// TwinCAT 3 PLC project lfe_optics
// Title: lcls-plc-lfe-optics
// Company: SLAC
// ProjectVersion: 4.0.0
// ProgramVersion: 3.1.4022.7
// CompilerDefines: L
// libraries:
//   LCLS General, * (SLAC)
//   lcls2-cc-lib, * (SLAC)
//   Tc2_ControllerToolbox, * (Beckhoff Automation GmbH)
//   Tc2_MC2, * (Beckhoff Automation GmbH)
//   Tc2_SerialCom, * (Beckhoff Automation GmbH)
//   Tc2_Standard, * (Beckhoff Automation GmbH)
//   Tc2_System, * (Beckhoff Automation GmbH)
//   Tc2_Utilities, * (Beckhoff Automation GmbH)
//   Tc3_Module, * (Beckhoff Automation GmbH)
//   VisuDialogs, * (System)
//   lcls-twincat-motion,4.0.9,SLAC
//   lcls-twincat-optics,0.7.0,SLAC
//   PMPS,3.3.0,SLAC - LCLS
// project tree:
//   DUTs/ E_MR1L0_CoatingStates.TcDUT, E_MR2L0_CoatingStates.TcDUT
//   Version/ Global_Version.TcGVL
//   / GlobalTextList.TcGTLO (not stored), PiezoDriver.TcTTO, PlcTask.TcTTO, SerialIO.TcTTO (not stored), Visualization Manager.TcVMO (not stored)
//   GVLs/ GVL_COM_Buffers.TcGVL, GVL_M1L0.TcGVL, GVL_M1L0_Constants.TcGVL, GVL_M2L0.TcGVL, GVL_M2L0_Constants.TcGVL, GVL_PMPS.TcGVL, GVL_SerialIO.TcGVL, GVL_States.TcGVL
//   POUs/ Main.TcPOU, PRG_1_PlcTask.TcPOU, PRG_MR1L0_HOMS.TcPOU, PRG_MR2L0_HOMS.TcPOU, PRG_PMPS.TcPOU, PRG_SP1L0_DCCM.TcPOU, P_CoatingProtections.TcPOU
//   POUs/Serial Comm/ PiezoSerial.TcPOU, P_Serial_Com.TcPOU
// real-time tasks:
//   TASK PlcTask: cycle T#10ms, priority 20, ADS port 350
//   TASK PiezoDriver: cycle T#1ms, priority 3, ADS port 351
//   TASK SerialIO: cycle T#2ms, priority 1, ADS port 352
// motion (NC):
//   TASK NC-Task 1 SAF: cycle T#2ms, priority 4, ADS port 501
//   TASK NC-Task 1 SVB: cycle T#10ms, priority 8, ADS port 511
//   AXIS M1L0-Yup (id 1)
//     General: UnitName=um
//     Dynamic: Acceleration=200, Deceleration=200, DelayTime=0.008
//     Velo: Maximum=200
//     OtherSettings: AllowMotionCmdToSlave=true
//     encoder EncType=29
//       EncPara: ScaleFactorNumerator=0.001, Offset=-16171.8, MaxCount=#xffffffff, ReferenceSystem=1
//         SoftEndMinControl: Enable=true, Range=-12605.3
//         SoftEndMaxControl: Enable=true, Range=10852.77
//         Inc: RefSoftSyncMask=#x0000ffff
//     drive DrvType=24
//       DrvPara: Inverse=true
//         Analog: VeloReferenz=488.28125, ScaleFactorActTorque=0.1
//         TimeComp: TaskDelayCycles=1
//     controller CtrType=2
//       CtrPara: PriorControlFactor=1
//         PosDiffControl: Range=100
//         PID: PosKp=50, PosExtKp=10, DeadBandPosition=0.3
//         Observer: BandWidth=20
//   AXIS M1L0-Ydwn (id 2)
//     General: UnitName=um
//     Dynamic: Acceleration=200, Deceleration=200, DelayTime=0.008
//     Velo: Maximum=200
//     OtherSettings: AllowMotionCmdToSlave=true
//     encoder EncType=29
//       EncPara: ScaleFactorNumerator=0.001, Offset=-14866.9, MaxCount=#xffffffff, ReferenceSystem=1
//         SoftEndMinControl: Enable=true, Range=-12700.5
//         SoftEndMaxControl: Enable=true, Range=10957.45
//         Inc: RefSoftSyncMask=#x0000ffff
//     drive DrvType=24
//       DrvPara: Inverse=true
//         Analog: VeloReferenz=488.28125, ScaleFactorActTorque=0.1
//         TimeComp: TaskDelayCycles=1
//     controller CtrType=2
//       CtrPara: PriorControlFactor=1
//         PosDiffControl: Range=100
//         PID: PosKp=50, PosExtKp=10, DeadBandPosition=0.3
//         Observer: BandWidth=20
//   AXIS M1L0-Xup (id 3)
//     General: UnitName=um
//     Dynamic: Acceleration=2000, Deceleration=2000, DelayTime=0.008
//     Velo: Maximum=1000
//     OtherSettings: AllowMotionCmdToSlave=true
//     encoder EncType=29
//       EncPara: ScaleFactorNumerator=0.001, Offset=-24797.788, MaxCount=#xffffffff, ReferenceSystem=1
//         SoftEndMinControl: Enable=true, Range=-600
//         SoftEndMaxControl: Enable=true, Range=690
//         Inc: RefSoftSyncMask=#x0000ffff
//     drive DrvType=24
//       Analog: VeloReferenz=1220.703125, ScaleFactorActTorque=0.1
//       TimeComp: TaskDelayCycles=1
//     controller CtrType=2
//       CtrPara: PriorControlFactor=1
//         PosDiffControl: Range=100
//         PID: PosKp=50, PosExtKp=50, DeadBandPosition=0.4
//         Observer: BandWidth=20
//   AXIS M1L0-Xdwn (id 4)
//     General: UnitName=um
//     Dynamic: Acceleration=2000, Deceleration=2000, DelayTime=0.008
//     Velo: Maximum=1000
//     OtherSettings: AllowMotionCmdToSlave=true
//     encoder EncType=29
//       EncPara: ScaleFactorNumerator=0.001, Offset=-22825.528, MaxCount=#xffffffff, ReferenceSystem=1
//         SoftEndMinControl: Enable=true, Range=-600
//         SoftEndMaxControl: Enable=true, Range=690
//         Inc: RefSoftSyncMask=#x0000ffff
//     drive DrvType=24
//       DrvPara: Inverse=true
//         Analog: VeloReferenz=1220.703125, ScaleFactorActTorque=0.1
//         TimeComp: TaskDelayCycles=1
//     controller CtrType=2
//       CtrPara: PriorControlFactor=1
//         PosDiffControl: Range=100
//         PID: PosKp=50, PosExtKp=50, DeadBandPosition=0.4
//         Observer: BandWidth=20
//   AXIS M1L0-Pitch (id 5)
//     General: UnitName=urad
//     Dynamic: Acceleration=390, Deceleration=390, DelayTime=0.008
//     Velo: Maximum=150
//     OtherSettings: AllowMotionCmdToSlave=true
//     encoder EncType=29
//       EncPara: ScaleFactorNumerator=0.001949317739, Offset=-16765.03, MaxCount=#xffffffff, ReferenceSystem=1
//         FilterTime: TPos=0.2
//         SoftEndMinControl: Enable=true, Range=-182
//         SoftEndMaxControl: Enable=true, Range=120
//         Inc: RefSoftSyncMask=#x0000ffff
//     drive DrvType=24
//       Analog: VeloReferenz=371.8, ScaleFactorActTorque=0.1
//       TimeComp: TaskDelayCycles=1
//     controller CtrType=2
//       CtrPara: PriorControlFactor=1
//         PosDiffControl: Range=20
//         PID: PosKp=2, PosExtKp=1, DeadBandPosition=0.01
//         Observer: BandWidth=20
//   AXIS M1L0-Bender (id 6)
//     General: UnitName=um
//     Dynamic: Acceleration=150, Deceleration=150, DelayTime=0.008
//     Velo: Maximum=150
//     OtherSettings: AllowMotionCmdToSlave=true
//     encoder EncType=29
//       EncPara: ScaleFactorNumerator=0.001, Offset=-4270000.1, MaxCount=#xffffffff, ReferenceSystem=1
//         SoftEndMinControl: Enable=true, Range=-1100.1
//         SoftEndMaxControl: Enable=true, Range=8149.9
//         Inc: RefSoftSyncMask=#x0000ffff
//     drive DrvType=24
//       DrvPara: Inverse=true
//         Analog: VeloReferenz=195.3125, ScaleFactorActTorque=0.1
//         TimeComp: TaskDelayCycles=1
//     controller CtrType=2
//       CtrPara: PriorControlFactor=1
//         PID: PosKp=10, PosExtKp=0.001, PosExtVelo=0.9, DeadBandPosition=0.1
//         Observer: BandWidth=20
//   AXIS M2L0-Yup (id 7)
//     General: UnitName=um
//     Dynamic: Acceleration=200, Deceleration=200, DelayTime=0.008
//     Velo: Maximum=200
//     OtherSettings: AllowMotionCmdToSlave=true
//     encoder EncType=29
//       EncPara: ScaleFactorNumerator=0.001, Offset=-12018.2, MaxCount=#xffffffff, MaxCountHighDWord=#x0000001f
//         SoftEndMinControl: Enable=true, Range=-9518.2
//         SoftEndMaxControl: Enable=true, Range=7519.8
//         Inc: RefSoftSyncMask=#x0000ffff
//     drive DrvType=24
//       DrvPara: Inverse=true
//         Analog: VeloReferenz=488.28125, ScaleFactorActTorque=0.1
//         TimeComp: TaskDelayCycles=1
//     controller CtrType=2
//       CtrPara: PriorControlFactor=1
//         PosDiffControl: Range=100
//         PID: PosKp=20, PosExtKp=5, DeadBandPosition=0.4
//         Observer: BandWidth=20
//   AXIS M2L0-Ydwn (id 8)
//     General: UnitName=um
//     Dynamic: Acceleration=200, Deceleration=200, DelayTime=0.008
//     Velo: Maximum=200
//     OtherSettings: AllowMotionCmdToSlave=true
//     encoder EncType=29
//       EncPara: ScaleFactorNumerator=0.001, Offset=-15143.7, MaxCount=#xffffffff, MaxCountHighDWord=#x0000001f
//         SoftEndMinControl: Enable=true, Range=-9987.7
//         SoftEndMaxControl: Enable=true, Range=7561.3
//         Inc: RefSoftSyncMask=#x0000ffff
//     drive DrvType=24
//       DrvPara: Inverse=true
//         Analog: VeloReferenz=488.28125, ScaleFactorActTorque=0.1
//         TimeComp: TaskDelayCycles=1
//     controller CtrType=2
//       CtrPara: PriorControlFactor=1
//         PosDiffControl: Range=100
//         PID: PosKp=20, PosExtKp=5, DeadBandPosition=0.4
//         Observer: BandWidth=20
//   AXIS M2L0-Xup (id 9)
//     General: UnitName=um
//     Dynamic: Acceleration=2000, Deceleration=2000, DelayTime=0.008
//     Velo: Maximum=1000
//     OtherSettings: AllowMotionCmdToSlave=true
//     encoder EncType=29
//       EncPara: ScaleFactorNumerator=0.001, Offset=-25363.4, MaxCount=#xffffffff, MaxCountHighDWord=#x0000001f
//         SoftEndMinControl: Enable=true, Range=-1063.4
//         SoftEndMaxControl: Enable=true, Range=1000
//         Inc: RefSoftSyncMask=#x0000ffff
//     drive DrvType=24
//       Analog: VeloReferenz=1220.703125, ScaleFactorActTorque=0.1
//       TimeComp: TaskDelayCycles=1
//     controller CtrType=2
//       CtrPara: PriorControlFactor=1
//         PosDiffControl: Range=100
//         PID: PosKp=10, PosExtKp=1, DeadBandPosition=0.4
//         Observer: BandWidth=20
//   AXIS M2L0-Xdwn (id 10)
//     General: UnitName=um
//     Dynamic: Acceleration=2000, Deceleration=2000, DelayTime=0.008
//     Velo: Maximum=1000
//     OtherSettings: AllowMotionCmdToSlave=true
//     encoder EncType=29
//       EncPara: ScaleFactorNumerator=0.001, Offset=-24398.1, MaxCount=#xffffffff, MaxCountHighDWord=#x0000001f
//         SoftEndMinControl: Enable=true, Range=-1289.2
//         SoftEndMaxControl: Enable=true, Range=1100.1
//         Inc: RefSoftSyncMask=#x0000ffff
//     drive DrvType=24
//       DrvPara: Inverse=true
//         Analog: VeloReferenz=1220.703125, ScaleFactorActTorque=0.1
//         TimeComp: TaskDelayCycles=1
//     controller CtrType=2
//       CtrPara: PriorControlFactor=1
//         PosDiffControl: Range=100
//         PID: PosKp=10, PosExtKp=1, DeadBandPosition=0.4
//         Observer: BandWidth=20
//   AXIS M2L0-Pitch (id 11)
//     General: UnitName=urad
//     Dynamic: Acceleration=390, Deceleration=390
//     Velo: Maximum=150
//     OtherSettings: AllowMotionCmdToSlave=true
//     encoder EncType=29
//       EncPara: ScaleFactorNumerator=0.001949317739, Offset=-18462.6, MaxCount=#xffffffff, MaxCountHighDWord=#x0000001f
//         FilterTime: TPos=0.2
//         SoftEndMinControl: Enable=true, Range=-45.1
//         SoftEndMaxControl: Enable=true, Range=154.9
//         Inc: RefSoftSyncMask=#x0000ffff
//     drive DrvType=24
//       Analog: VeloReferenz=371.8, ScaleFactorActTorque=0.1
//       TimeComp: TaskDelayCycles=1
//     controller CtrType=2
//       CtrPara: PriorControlFactor=1
//         PosDiffControl: Range=20
//         PID: PosKp=2, PosExtKp=1, DeadBandPosition=0.01
//         Observer: BandWidth=20
//   AXIS M2L0-Bender (id 12)
//     General: UnitName=um
//     Dynamic: Acceleration=150, Deceleration=150, DelayTime=0.008
//     Velo: Maximum=150
//     OtherSettings: AllowMotionCmdToSlave=true
//     encoder EncType=29
//       EncPara: ScaleFactorNumerator=0.001, Offset=-4268979, MaxCount=#xffffffff
//         SoftEndMinControl: Enable=true, Range=-2
//         SoftEndMaxControl: Enable=true, Range=10762
//         Inc: RefSoftSyncMask=#x0000ffff
//     drive DrvType=24
//       DrvPara: Inverse=true
//         Analog: VeloReferenz=195.3125, ScaleFactorActTorque=0.1
//         TimeComp: TaskDelayCycles=1
//     controller CtrType=2
//       CtrPara: PriorControlFactor=1
//         PID: PosKp=10, PosExtKp=0.001, PosExtVelo=0.9, DeadBandPosition=0.1
//         Observer: BandWidth=20
//   AXIS SP1L0-TH1 (id 13)
//     General: UnitName=Degree
//     Dynamic: AccelerationMaximum=10, DecelerationMaximum=10, Acceleration=8.99313, Deceleration=8.99313, Jerk=27.7544, DelayTime=0.008
//     Velo: SlowManual=1, FastManual=2, Maximum=0.12
//     TargetPosControl: Range=0.001
//     OtherSettings: AllowMotionCmdToSlave=true, PulseDistancePos=0.5, PulseDistanceNeg=0.5
//     encoder EncType=29
//       EncPara: ScaleFactorNumerator=5.72957795, ScaleFactorDenominator=10000000, Offset=-11, MaxCount=#xffffffff, MaxCountHighDWord=#x0000001f
//         SoftEndMinControl: Enable=true, Range=-1
//         SoftEndMaxControl: Enable=true, Range=71
//         Inc: RefSoftSyncMask=#x0000ffff
//     drive DrvType=24
//       Analog: VeloReferenz=0.1275, TorqueSetpointScale=10, ScaleFactorActTorque=0.1
//       TimeComp: TaskDelayCycles=1
//     controller CtrType=3
//       CtrPara: PriorControlFactor=1
//         PosDiffControl: Range=0.05
//         PID: PosKp=10, PosTv=0.2, DeadBandPosition=0.0001
//         Observer: BandWidth=20
//   AXIS SP1L0-TH2 (id 14)
//     General: UnitName=Degree
//     Dynamic: AccelerationMaximum=10, DecelerationMaximum=10, Acceleration=9, Deceleration=9, Jerk=27.7, DelayTime=0.008
//     Velo: SlowManual=0.1, FastManual=0.3, Maximum=0.12
//     PositionAreaControl: Range=0.05
//     TargetPosControl: Range=0.0001
//     OtherSettings: AllowMotionCmdToSlave=true
//     encoder EncType=29
//       EncPara: ScaleFactorNumerator=5.72957795, ScaleFactorDenominator=10000000, Offset=-10.66, MaxCount=#xffffffff, MaxCountHighDWord=#x0000001f
//         SoftEndMinControl: Enable=true, Range=-1
//         SoftEndMaxControl: Enable=true, Range=71
//         Inc: RefSoftSyncMask=#x0000ffff
//     drive DrvType=24
//       DrvPara: Inverse=true
//         Analog: VeloReferenz=0.127500425, TorqueSetpointScale=10, ScaleFactorActTorque=0.1
//         TimeComp: TaskDelayCycles=1
//     controller CtrType=3
//       CtrPara: PriorControlFactor=1
//         PosDiffControl: Range=0.05
//         PID: PosKp=10, PosTv=0.2, DeadBandPosition=0.0001
//         Observer: BandWidth=20
//   AXIS SP1L0-Tx (id 15)
//     Dynamic: AccelerationMaximum=20, DecelerationMaximum=20, Acceleration=10, Deceleration=10, Jerk=100, DelayTime=0.008
//     Velo: SlowManual=0.3, FastManual=1, Maximum=1
//     PositionAreaControl: Range=0.2
//     TargetPosControl: Range=0.0005
//     OtherSettings: AllowMotionCmdToSlave=true, PulseDistancePos=1, PulseDistanceNeg=1
//     encoder EncType=29
//       EncPara: ScaleFactorNumerator=50, ScaleFactorDenominator=1000000, Offset=-29.5, MaxCount=#xffffffff, MaxCountHighDWord=#x0000001f
//         SoftEndMinControl: Enable=true, Range=-13
//         SoftEndMaxControl: Enable=true, Range=3
//         Inc: RefSoftSyncMask=#x0000ffff
//     drive DrvType=24
//       Analog: VeloReferenz=1, TorqueSetpointScale=10, ScaleFactorActTorque=0.1
//       TimeComp: TaskDelayCycles=1
//     controller CtrType=3
//       CtrPara: PriorControlFactor=1
//         PosDiffControl: Range=0.1
//         PID: PosKp=10, PosTv=0.2, DeadBandPosition=0.0001
//         Observer: BandWidth=20
//   AXIS SP1L0-Txd (id 16)
//     Dynamic: AccelerationMaximum=20, DecelerationMaximum=20, Acceleration=10, Deceleration=10, Jerk=100, DelayTime=0.008
//     Velo: SlowManual=0.075, FastManual=0.2, Maximum=2
//     PositionAreaControl: Range=0.01
//     TargetPosControl: Range=0.0001
//     OtherSettings: AllowMotionCmdToSlave=true, PulseDistancePos=0.05, PulseDistanceNeg=0.05
//     encoder EncType=29
//       EncPara: ScaleFactorNumerator=50, ScaleFactorDenominator=1000000, Offset=-6871908.2, MaxCount=#xffffffff, MaxCountHighDWord=#x0000001f
//         SoftEndMinControl: Enable=true, Range=-12
//         SoftEndMaxControl: Enable=true, Range=12
//         Inc: RefSoftSyncMask=#x0000ffff
//     drive DrvType=24
//       DrvPara: Inverse=true
//         Analog: VeloReferenz=10.668, TorqueSetpointScale=10, ScaleFactorActTorque=0.1
//         TimeComp: TaskDelayCycles=1
//     controller CtrType=3
//       CtrPara: PriorControlFactor=1
//         PosDiffControl: Range=0.15
//         PID: PosKp=4, PosTv=0.2, PosTd=1, DeadBandPosition=0.0001
//         Observer: BandWidth=20
//   AXIS SP1L0-Tyd (id 17)
//     Dynamic: AccelerationMaximum=20, DecelerationMaximum=20, Acceleration=10, Deceleration=10, Jerk=100, DelayTime=0.008
//     Velo: SlowManual=0.5, FastManual=1, Maximum=2
//     PositionAreaControl: Range=0.05
//     TargetPosControl: Range=0.05
//     OtherSettings: AllowMotionCmdToSlave=true
//     encoder EncType=29
//       EncPara: ScaleFactorNumerator=50, ScaleFactorDenominator=1000000, Offset=-6871872.92, MaxCount=#xffffffff, MaxCountHighDWord=#x0000001f
//         SoftEndMaxControl: Range=48
//         Inc: RefSoftSyncMask=#x0000ffff
//     drive DrvType=24
//       Analog: VeloReferenz=12.6999, TorqueSetpointScale=10, ScaleFactorActTorque=0.1
//       TimeComp: TaskDelayCycles=1
//     controller CtrType=3
//       CtrPara: PriorControlFactor=1
//         PosDiffControl: Range=0.25
//         PID: PosKp=15, PosTv=0.2, DeadBandPosition=0.01
//         Observer: BandWidth=20
// I/O:
//   DEVICE Device 1 (EtherCAT), AmsNetId 172.21.88.30.2.1
//     Term 1 (EK1200) [EK1200-5000 EtherCAT Power supply (2A E-Bus)]
//       PMPS_FFO
//       Term 3 (EL6070) [EL6070 1Ch. Licensing-Terminal]
//       PMPS_PRE [EL6695 EtherCAT Bridge terminal (Primary)]
//       Term 5 (EK1122) [EK1122 2 port EtherCAT junction]
//         Box 6 (CU1124) [CU1124 EtherCAT junction (4-ports)]
//           EK1100_SP1L0 [EK1100 EtherCAT Coupler (2A E-Bus)]
//             EL7047_SP1L0_th1 [EL7047 1Ch. Stepper motor output stage (50V, 5A)]
//             EL7047_SP1L0_th2 [EL7047 1Ch. Stepper motor output stage (50V, 5A)]
//             EL7047_SP1L0_tx [EL7047 1Ch. Stepper motor output stage (50V, 5A)]
//             EL7047_SP1L0_txd [EL7047 1Ch. Stepper motor output stage (50V, 5A)]
//             EL7047_SP1L0_tyd [EL7047 1Ch. Stepper motor output stage (50V, 5A)]
//             EL5042_SP1L0_th1_th2 [EL5042 2Ch. BiSS-C Encoder]
//             EL5042_SP1L0_tx_txd [EL5042 2Ch. BiSS-C Encoder]
//             EL5042_SP1L0_tyd [EL5042 2Ch. BiSS-C Encoder]
//             EL1008_SP1L0_STO_DI [EL1008 8Ch. Dig. Input 24V, 3ms]
//             EL2008_SP1L0_DO [EL2008 8Ch. Dig. Output 24V, 0.5A]
//             EL3054_SP1L0_AI [EL3054 4Ch. Ana. Input 4-20mA]
//             EL9011_SP1L0 [EL9011 End Terminal]
//           EK1100_M2L0 [EK1100 EtherCAT Coupler (2A E-Bus)]
//             EL7041-1000_M2L0_Xup [EL7041-1000 1Ch. Stepper motor output stage (50V, 5A, standard)]
//             EL7041-1000_M2L0_Xdwn [EL7041-1000 1Ch. Stepper motor output stage (50V, 5A, standard)]
//             EL7041-1000_M2L0_Yup [EL7041-1000 1Ch. Stepper motor output stage (50V, 5A, standard)]
//             EL7041-1000_M2L0_Ydwn [EL7041-1000 1Ch. Stepper motor output stage (50V, 5A, standard)]
//             EL7041-1000_M2L0_PitchCoarse [EL7041-1000 1Ch. Stepper motor output stage (50V, 5A, standard)]
//             EL7041-1000_M2L0_Bender [EL7041-1000 1Ch. Stepper motor output stage (50V, 5A, standard)]
//             EL6001_M2L0_PitchFine [EL6001 Interface (RS232)]
//             EL5042_M2L0_Xupdwn [EL5042 2Ch. BiSS-C Encoder]
//             EL5042_M2L0_Yupdwn [EL5042 2Ch. BiSS-C Encoder]
//             EL5042_M2L0_PitchBender [EL5042 2Ch. BiSS-C Encoder]
//             EL1004_M2L0_STO [EL1004 4Ch. Dig. Input 24V, 3ms]
//             EL3054_M2L0_FWM_PRSM [EL3054 4Ch. Ana. Input 4-20mA]
//             EL9505_M2L0_BenderLims [EL9505 Power supply terminal 5V]
//             Term 33 (EL9011) [EL9011 End Terminal]
//           EP2008-0001_M1M2_VCV
//         EK1100_M1L0 [EK1100 EtherCAT Coupler (2A E-Bus)]
//           EL7041-1000_M1L0_Xup [EL7041-1000 1Ch. Stepper motor output stage (50V, 5A, standard)]
//           EL7041-1000_M1L0_Xdwn
//           EL7041-1000_M1L0_Yup [EL7041-1000 1Ch. Stepper motor output stage (50V, 5A, standard)]
//           EL7041-1000_M1L0_Ydwn [EL7041-1000 1Ch. Stepper motor output stage (50V, 5A, standard)]
//           EL7041-1000_M1L0_PitchCoarse [EL7041-1000 1Ch. Stepper motor output stage (50V, 5A, standard)]
//           EL7041-1000_M1L0_Bender
//           EL6001_M1L0_PitchFine
//           EL5042_M1L0_Xupdwn
//           EL5042_M1L0_Yupdwn
//           EL5042_M1L0_PitchBender [EL5042 2Ch. BiSS-C Encoder]
//           EL1004_M1L0_STO
//           EL3054_M1L0_FWM_PRSM
//           EL9505_M1L0_BenderLims
//           Term 32 (EL9011)
// variable links:
//   (this object) <-> Device 1 (EtherCAT)/Term 1 (EK1200)/Term 5 (EK1122)/EK1100_M1L0/EL5042_M1L0_Yupdwn
//     Enc/Inputs/In/nComState @bit 1 <-> WcState/InputToggle
//     Enc/Inputs/In/nComState <-> WcState/WcState
//     Enc/Inputs/In/nDataIn1 <-> FB Inputs Channel 1/Position
//     Enc/Inputs/In/nDataIn1 <-> FB Inputs Channel 2/Position
//     Enc/Inputs/In/nState1 @bit 12 <-> FB Inputs Channel 1/Status/Diag
//     Enc/Inputs/In/nState1 @bit 12 <-> FB Inputs Channel 2/Status/Diag
//     Enc/Inputs/In/nState1 @bit 1 <-> FB Inputs Channel 1/Status/Error
//     Enc/Inputs/In/nState1 @bit 1 <-> FB Inputs Channel 2/Status/Error
//     Enc/Inputs/In/nState1 @bit 14 <-> FB Inputs Channel 1/Status/Input cycle counter
//     Enc/Inputs/In/nState1 @bit 14 <-> FB Inputs Channel 2/Status/Input cycle counter
//     Enc/Inputs/In/nState1 @bit 2 <-> FB Inputs Channel 1/Status/Ready
//     Enc/Inputs/In/nState1 @bit 2 <-> FB Inputs Channel 2/Status/Ready
//     Enc/Inputs/In/nState1 @bit 13 <-> FB Inputs Channel 1/Status/TxPDO State
//     Enc/Inputs/In/nState1 @bit 13 <-> FB Inputs Channel 2/Status/TxPDO State
//     Enc/Inputs/In/nState1 <-> FB Inputs Channel 1/Status/Warning
//     Enc/Inputs/In/nState1 <-> FB Inputs Channel 2/Status/Warning
//   (this object) <-> Device 1 (EtherCAT)/Term 1 (EK1200)/Term 5 (EK1122)/EK1100_M1L0/EL7041-1000_M1L0_Yup
//     Drive/Inputs/In/nState1 @bit 3 <-> STM Status/Status/Error
//     Drive/Inputs/In/nState1 @bit 5 <-> STM Status/Status/Moving negative
//     Drive/Inputs/In/nState1 @bit 4 <-> STM Status/Status/Moving positive
//     Drive/Inputs/In/nState1 @bit 1 <-> STM Status/Status/Ready
//     Drive/Inputs/In/nState1 <-> STM Status/Status/Ready to enable
//     Drive/Inputs/In/nState1 @bit 6 <-> STM Status/Status/Torque reduced
//     Drive/Inputs/In/nState1 @bit 2 <-> STM Status/Status/Warning
//     Drive/Inputs/In/nState2 @bit 3 <-> STM Status/Status/Digital input 1
//     Drive/Inputs/In/nState2 @bit 4 <-> STM Status/Status/Digital input 2
//     Drive/Inputs/In/nState2 @bit 5 <-> STM Status/Status/Sync error
//     Drive/Inputs/In/nState2 @bit 7 <-> STM Status/Status/TxPDO Toggle
//     Drive/Inputs/In/nState4 @bit 1 <-> WcState/InputToggle
//     Drive/Inputs/In/nState4 <-> WcState/WcState
//     Drive/Outputs/Out/nCtrl1 <-> STM Control/Control/Enable
//     Drive/Outputs/Out/nCtrl1 @bit 2 <-> STM Control/Control/Reduce torque
//     Drive/Outputs/Out/nCtrl1 @bit 1 <-> STM Control/Control/Reset
//     Drive/Outputs/Out/nDataOut2[0] <-> STM Velocity/Velocity
//   (this object) <-> Device 1 (EtherCAT)/Term 1 (EK1200)/Term 5 (EK1122)/EK1100_M1L0/EL7041-1000_M1L0_Ydwn
//     Drive/Inputs/In/nState1 @bit 3 <-> STM Status/Status/Error
//     Drive/Inputs/In/nState1 @bit 5 <-> STM Status/Status/Moving negative
//     Drive/Inputs/In/nState1 @bit 4 <-> STM Status/Status/Moving positive
//     Drive/Inputs/In/nState1 @bit 1 <-> STM Status/Status/Ready
//     Drive/Inputs/In/nState1 <-> STM Status/Status/Ready to enable
//     Drive/Inputs/In/nState1 @bit 6 <-> STM Status/Status/Torque reduced
//     Drive/Inputs/In/nState1 @bit 2 <-> STM Status/Status/Warning
//     Drive/Inputs/In/nState2 @bit 3 <-> STM Status/Status/Digital input 1
//     Drive/Inputs/In/nState2 @bit 4 <-> STM Status/Status/Digital input 2
//     Drive/Inputs/In/nState2 @bit 5 <-> STM Status/Status/Sync error
//     Drive/Inputs/In/nState2 @bit 7 <-> STM Status/Status/TxPDO Toggle
//     Drive/Inputs/In/nState4 @bit 1 <-> WcState/InputToggle
//     Drive/Inputs/In/nState4 <-> WcState/WcState
//     Drive/Outputs/Out/nCtrl1 <-> STM Control/Control/Enable
//     Drive/Outputs/Out/nCtrl1 @bit 2 <-> STM Control/Control/Reduce torque
//     Drive/Outputs/Out/nCtrl1 @bit 1 <-> STM Control/Control/Reset
//     Drive/Outputs/Out/nDataOut2[0] <-> STM Velocity/Velocity
//   (this object) <-> Device 1 (EtherCAT)/Term 1 (EK1200)/Term 5 (EK1122)/EK1100_M1L0/EL5042_M1L0_Xupdwn
//     Enc/Inputs/In/nComState @bit 1 <-> WcState/InputToggle
//     Enc/Inputs/In/nComState <-> WcState/WcState
//     Enc/Inputs/In/nDataIn1 <-> FB Inputs Channel 1/Position
//     Enc/Inputs/In/nDataIn1 <-> FB Inputs Channel 2/Position
//     Enc/Inputs/In/nState1 @bit 12 <-> FB Inputs Channel 1/Status/Diag
//     Enc/Inputs/In/nState1 @bit 12 <-> FB Inputs Channel 2/Status/Diag
//     Enc/Inputs/In/nState1 @bit 1 <-> FB Inputs Channel 1/Status/Error
//     Enc/Inputs/In/nState1 @bit 1 <-> FB Inputs Channel 2/Status/Error
//     Enc/Inputs/In/nState1 @bit 14 <-> FB Inputs Channel 1/Status/Input cycle counter
//     Enc/Inputs/In/nState1 @bit 14 <-> FB Inputs Channel 2/Status/Input cycle counter
//     Enc/Inputs/In/nState1 @bit 2 <-> FB Inputs Channel 1/Status/Ready
//     Enc/Inputs/In/nState1 @bit 2 <-> FB Inputs Channel 2/Status/Ready
//     Enc/Inputs/In/nState1 @bit 13 <-> FB Inputs Channel 1/Status/TxPDO State
//     Enc/Inputs/In/nState1 @bit 13 <-> FB Inputs Channel 2/Status/TxPDO State
//     Enc/Inputs/In/nState1 <-> FB Inputs Channel 1/Status/Warning
//     Enc/Inputs/In/nState1 <-> FB Inputs Channel 2/Status/Warning
//   (this object) <-> Device 1 (EtherCAT)/Term 1 (EK1200)/Term 5 (EK1122)/EK1100_M1L0/EL7041-1000_M1L0_Xup
//     Drive/Inputs/In/nState1 @bit 3 <-> STM Status/Status/Error
//     Drive/Inputs/In/nState1 @bit 5 <-> STM Status/Status/Moving negative
//     Drive/Inputs/In/nState1 @bit 4 <-> STM Status/Status/Moving positive
//     Drive/Inputs/In/nState1 @bit 1 <-> STM Status/Status/Ready
//     Drive/Inputs/In/nState1 <-> STM Status/Status/Ready to enable
//     Drive/Inputs/In/nState1 @bit 6 <-> STM Status/Status/Torque reduced
//     Drive/Inputs/In/nState1 @bit 2 <-> STM Status/Status/Warning
//     Drive/Inputs/In/nState2 @bit 3 <-> STM Status/Status/Digital input 1
//     Drive/Inputs/In/nState2 @bit 4 <-> STM Status/Status/Digital input 2
//     Drive/Inputs/In/nState2 @bit 5 <-> STM Status/Status/Sync error
//     Drive/Inputs/In/nState2 @bit 7 <-> STM Status/Status/TxPDO Toggle
//     Drive/Inputs/In/nState4 @bit 1 <-> WcState/InputToggle
//     Drive/Inputs/In/nState4 <-> WcState/WcState
//     Drive/Outputs/Out/nCtrl1 <-> STM Control/Control/Enable
//     Drive/Outputs/Out/nCtrl1 @bit 2 <-> STM Control/Control/Reduce torque
//     Drive/Outputs/Out/nCtrl1 @bit 1 <-> STM Control/Control/Reset
//     Drive/Outputs/Out/nDataOut2[0] <-> STM Velocity/Velocity
//   (this object) <-> Device 1 (EtherCAT)/Term 1 (EK1200)/Term 5 (EK1122)/EK1100_M1L0/EL7041-1000_M1L0_Xdwn
//     Drive/Inputs/In/nState1 @bit 3 <-> STM Status/Status/Error
//     Drive/Inputs/In/nState1 @bit 5 <-> STM Status/Status/Moving negative
//     Drive/Inputs/In/nState1 @bit 4 <-> STM Status/Status/Moving positive
//     Drive/Inputs/In/nState1 @bit 1 <-> STM Status/Status/Ready
//     Drive/Inputs/In/nState1 <-> STM Status/Status/Ready to enable
//     Drive/Inputs/In/nState1 @bit 6 <-> STM Status/Status/Torque reduced
//     Drive/Inputs/In/nState1 @bit 2 <-> STM Status/Status/Warning
//     Drive/Inputs/In/nState2 @bit 3 <-> STM Status/Status/Digital input 1
//     Drive/Inputs/In/nState2 @bit 4 <-> STM Status/Status/Digital input 2
//     Drive/Inputs/In/nState2 @bit 5 <-> STM Status/Status/Sync error
//     Drive/Inputs/In/nState2 @bit 7 <-> STM Status/Status/TxPDO Toggle
//     Drive/Inputs/In/nState4 @bit 1 <-> WcState/InputToggle
//     Drive/Inputs/In/nState4 <-> WcState/WcState
//     Drive/Outputs/Out/nCtrl1 <-> STM Control/Control/Enable
//     Drive/Outputs/Out/nCtrl1 @bit 2 <-> STM Control/Control/Reduce torque
//     Drive/Outputs/Out/nCtrl1 @bit 1 <-> STM Control/Control/Reset
//     Drive/Outputs/Out/nDataOut2[0] <-> STM Velocity/Velocity
//   (this object) <-> Device 1 (EtherCAT)/Term 1 (EK1200)/Term 5 (EK1122)/EK1100_M1L0/EL5042_M1L0_PitchBender
//     Enc/Inputs/In/nComState @bit 1 <-> WcState/InputToggle
//     Enc/Inputs/In/nComState <-> WcState/WcState
//     Enc/Inputs/In/nDataIn1 <-> FB Inputs Channel 1/Position
//     Enc/Inputs/In/nDataIn1 <-> FB Inputs Channel 2/Position
//     Enc/Inputs/In/nState1 @bit 12 <-> FB Inputs Channel 1/Status/Diag
//     Enc/Inputs/In/nState1 @bit 12 <-> FB Inputs Channel 2/Status/Diag
//     Enc/Inputs/In/nState1 @bit 1 <-> FB Inputs Channel 1/Status/Error
//     Enc/Inputs/In/nState1 @bit 1 <-> FB Inputs Channel 2/Status/Error
//     Enc/Inputs/In/nState1 @bit 14 <-> FB Inputs Channel 1/Status/Input cycle counter
//     Enc/Inputs/In/nState1 @bit 14 <-> FB Inputs Channel 2/Status/Input cycle counter
//     Enc/Inputs/In/nState1 @bit 2 <-> FB Inputs Channel 1/Status/Ready
//     Enc/Inputs/In/nState1 @bit 2 <-> FB Inputs Channel 2/Status/Ready
//     Enc/Inputs/In/nState1 @bit 13 <-> FB Inputs Channel 1/Status/TxPDO State
//     Enc/Inputs/In/nState1 @bit 13 <-> FB Inputs Channel 2/Status/TxPDO State
//     Enc/Inputs/In/nState1 <-> FB Inputs Channel 1/Status/Warning
//     Enc/Inputs/In/nState1 <-> FB Inputs Channel 2/Status/Warning
//   (this object) <-> Device 1 (EtherCAT)/Term 1 (EK1200)/Term 5 (EK1122)/EK1100_M1L0/EL7041-1000_M1L0_PitchCoarse
//     Drive/Inputs/In/nState1 @bit 3 <-> STM Status/Status/Error
//     Drive/Inputs/In/nState1 @bit 5 <-> STM Status/Status/Moving negative
//     Drive/Inputs/In/nState1 @bit 4 <-> STM Status/Status/Moving positive
//     Drive/Inputs/In/nState1 @bit 1 <-> STM Status/Status/Ready
//     Drive/Inputs/In/nState1 <-> STM Status/Status/Ready to enable
//     Drive/Inputs/In/nState1 @bit 6 <-> STM Status/Status/Torque reduced
//     Drive/Inputs/In/nState1 @bit 2 <-> STM Status/Status/Warning
//     Drive/Inputs/In/nState2 @bit 3 <-> STM Status/Status/Digital input 1
//     Drive/Inputs/In/nState2 @bit 4 <-> STM Status/Status/Digital input 2
//     Drive/Inputs/In/nState2 @bit 5 <-> STM Status/Status/Sync error
//     Drive/Inputs/In/nState2 @bit 7 <-> STM Status/Status/TxPDO Toggle
//     Drive/Inputs/In/nState4 @bit 1 <-> WcState/InputToggle
//     Drive/Inputs/In/nState4 <-> WcState/WcState
//     Drive/Outputs/Out/nCtrl1 <-> STM Control/Control/Enable
//     Drive/Outputs/Out/nCtrl1 @bit 2 <-> STM Control/Control/Reduce torque
//     Drive/Outputs/Out/nCtrl1 @bit 1 <-> STM Control/Control/Reset
//     Drive/Outputs/Out/nDataOut2[0] <-> STM Velocity/Velocity
//   (this object) <-> Device 1 (EtherCAT)/Term 1 (EK1200)/Term 5 (EK1122)/EK1100_M1L0/EL7041-1000_M1L0_Bender
//     Drive/Inputs/In/nState1 @bit 3 <-> STM Status/Status/Error
//     Drive/Inputs/In/nState1 @bit 5 <-> STM Status/Status/Moving negative
//     Drive/Inputs/In/nState1 @bit 4 <-> STM Status/Status/Moving positive
//     Drive/Inputs/In/nState1 @bit 1 <-> STM Status/Status/Ready
//     Drive/Inputs/In/nState1 <-> STM Status/Status/Ready to enable
//     Drive/Inputs/In/nState1 @bit 6 <-> STM Status/Status/Torque reduced
//     Drive/Inputs/In/nState1 @bit 2 <-> STM Status/Status/Warning
//     Drive/Inputs/In/nState2 @bit 3 <-> STM Status/Status/Digital input 1
//     Drive/Inputs/In/nState2 @bit 4 <-> STM Status/Status/Digital input 2
//     Drive/Inputs/In/nState2 @bit 5 <-> STM Status/Status/Sync error
//     Drive/Inputs/In/nState2 @bit 7 <-> STM Status/Status/TxPDO Toggle
//     Drive/Inputs/In/nState4 @bit 1 <-> WcState/InputToggle
//     Drive/Inputs/In/nState4 <-> WcState/WcState
//     Drive/Outputs/Out/nCtrl1 <-> STM Control/Control/Enable
//     Drive/Outputs/Out/nCtrl1 @bit 2 <-> STM Control/Control/Reduce torque
//     Drive/Outputs/Out/nCtrl1 @bit 1 <-> STM Control/Control/Reset
//     Drive/Outputs/Out/nDataOut2[0] <-> STM Velocity/Velocity
//   (this object) <-> Device 1 (EtherCAT)/Term 1 (EK1200)/Term 5 (EK1122)/Box 6 (CU1124)/EK1100_M2L0/EL5042_M2L0_Yupdwn
//     Enc/Inputs/In/nComState @bit 1 <-> WcState/InputToggle
//     Enc/Inputs/In/nComState <-> WcState/WcState
//     Enc/Inputs/In/nDataIn1 <-> FB Inputs Channel 1/Position
//     Enc/Inputs/In/nDataIn1 <-> FB Inputs Channel 2/Position
//     Enc/Inputs/In/nState1 @bit 12 <-> FB Inputs Channel 1/Status/Diag
//     Enc/Inputs/In/nState1 @bit 12 <-> FB Inputs Channel 2/Status/Diag
//     Enc/Inputs/In/nState1 @bit 1 <-> FB Inputs Channel 1/Status/Error
//     Enc/Inputs/In/nState1 @bit 1 <-> FB Inputs Channel 2/Status/Error
//     Enc/Inputs/In/nState1 @bit 14 <-> FB Inputs Channel 1/Status/Input cycle counter
//     Enc/Inputs/In/nState1 @bit 14 <-> FB Inputs Channel 2/Status/Input cycle counter
//     Enc/Inputs/In/nState1 @bit 2 <-> FB Inputs Channel 1/Status/Ready
//     Enc/Inputs/In/nState1 @bit 2 <-> FB Inputs Channel 2/Status/Ready
//     Enc/Inputs/In/nState1 @bit 13 <-> FB Inputs Channel 1/Status/TxPDO State
//     Enc/Inputs/In/nState1 @bit 13 <-> FB Inputs Channel 2/Status/TxPDO State
//     Enc/Inputs/In/nState1 <-> FB Inputs Channel 1/Status/Warning
//     Enc/Inputs/In/nState1 <-> FB Inputs Channel 2/Status/Warning
//   (this object) <-> Device 1 (EtherCAT)/Term 1 (EK1200)/Term 5 (EK1122)/Box 6 (CU1124)/EK1100_M2L0/EL7041-1000_M2L0_Yup
//     Drive/Inputs/In/nState1 @bit 3 <-> STM Status/Status/Error
//     Drive/Inputs/In/nState1 @bit 5 <-> STM Status/Status/Moving negative
//     Drive/Inputs/In/nState1 @bit 4 <-> STM Status/Status/Moving positive
//     Drive/Inputs/In/nState1 @bit 1 <-> STM Status/Status/Ready
//     Drive/Inputs/In/nState1 <-> STM Status/Status/Ready to enable
//     Drive/Inputs/In/nState1 @bit 6 <-> STM Status/Status/Torque reduced
//     Drive/Inputs/In/nState1 @bit 2 <-> STM Status/Status/Warning
//     Drive/Inputs/In/nState2 @bit 3 <-> STM Status/Status/Digital input 1
//     Drive/Inputs/In/nState2 @bit 4 <-> STM Status/Status/Digital input 2
//     Drive/Inputs/In/nState2 @bit 5 <-> STM Status/Status/Sync error
//     Drive/Inputs/In/nState2 @bit 7 <-> STM Status/Status/TxPDO Toggle
//     Drive/Inputs/In/nState4 @bit 1 <-> WcState/InputToggle
//     Drive/Inputs/In/nState4 <-> WcState/WcState
//     Drive/Outputs/Out/nCtrl1 <-> STM Control/Control/Enable
//     Drive/Outputs/Out/nCtrl1 @bit 2 <-> STM Control/Control/Reduce torque
//     Drive/Outputs/Out/nCtrl1 @bit 1 <-> STM Control/Control/Reset
//     Drive/Outputs/Out/nDataOut2[0] <-> STM Velocity/Velocity
//   (this object) <-> Device 1 (EtherCAT)/Term 1 (EK1200)/Term 5 (EK1122)/Box 6 (CU1124)/EK1100_M2L0/EL7041-1000_M2L0_Ydwn
//     Drive/Inputs/In/nState1 @bit 3 <-> STM Status/Status/Error
//     Drive/Inputs/In/nState1 @bit 5 <-> STM Status/Status/Moving negative
//     Drive/Inputs/In/nState1 @bit 4 <-> STM Status/Status/Moving positive
//     Drive/Inputs/In/nState1 @bit 1 <-> STM Status/Status/Ready
//     Drive/Inputs/In/nState1 <-> STM Status/Status/Ready to enable
//     Drive/Inputs/In/nState1 @bit 6 <-> STM Status/Status/Torque reduced
//     Drive/Inputs/In/nState1 @bit 2 <-> STM Status/Status/Warning
//     Drive/Inputs/In/nState2 @bit 3 <-> STM Status/Status/Digital input 1
//     Drive/Inputs/In/nState2 @bit 4 <-> STM Status/Status/Digital input 2
//     Drive/Inputs/In/nState2 @bit 5 <-> STM Status/Status/Sync error
//     Drive/Inputs/In/nState2 @bit 7 <-> STM Status/Status/TxPDO Toggle
//     Drive/Inputs/In/nState4 @bit 1 <-> WcState/InputToggle
//     Drive/Inputs/In/nState4 <-> WcState/WcState
//     Drive/Outputs/Out/nCtrl1 <-> STM Control/Control/Enable
//     Drive/Outputs/Out/nCtrl1 @bit 2 <-> STM Control/Control/Reduce torque
//     Drive/Outputs/Out/nCtrl1 @bit 1 <-> STM Control/Control/Reset
//     Drive/Outputs/Out/nDataOut2[0] <-> STM Velocity/Velocity
//   (this object) <-> Device 1 (EtherCAT)/Term 1 (EK1200)/Term 5 (EK1122)/Box 6 (CU1124)/EK1100_M2L0/EL5042_M2L0_Xupdwn
//     Enc/Inputs/In/nComState @bit 1 <-> WcState/InputToggle
//     Enc/Inputs/In/nComState <-> WcState/WcState
//     Enc/Inputs/In/nDataIn1 <-> FB Inputs Channel 1/Position
//     Enc/Inputs/In/nDataIn1 <-> FB Inputs Channel 2/Position
//     Enc/Inputs/In/nState1 @bit 12 <-> FB Inputs Channel 1/Status/Diag
//     Enc/Inputs/In/nState1 @bit 12 <-> FB Inputs Channel 2/Status/Diag
//     Enc/Inputs/In/nState1 @bit 1 <-> FB Inputs Channel 1/Status/Error
//     Enc/Inputs/In/nState1 @bit 1 <-> FB Inputs Channel 2/Status/Error
//     Enc/Inputs/In/nState1 @bit 14 <-> FB Inputs Channel 1/Status/Input cycle counter
//     Enc/Inputs/In/nState1 @bit 14 <-> FB Inputs Channel 2/Status/Input cycle counter
//     Enc/Inputs/In/nState1 @bit 2 <-> FB Inputs Channel 1/Status/Ready
//     Enc/Inputs/In/nState1 @bit 2 <-> FB Inputs Channel 2/Status/Ready
//     Enc/Inputs/In/nState1 @bit 13 <-> FB Inputs Channel 1/Status/TxPDO State
//     Enc/Inputs/In/nState1 @bit 13 <-> FB Inputs Channel 2/Status/TxPDO State
//     Enc/Inputs/In/nState1 <-> FB Inputs Channel 1/Status/Warning
//     Enc/Inputs/In/nState1 <-> FB Inputs Channel 2/Status/Warning
//   (this object) <-> Device 1 (EtherCAT)/Term 1 (EK1200)/Term 5 (EK1122)/Box 6 (CU1124)/EK1100_M2L0/EL7041-1000_M2L0_Xup
//     Drive/Inputs/In/nState1 @bit 3 <-> STM Status/Status/Error
//     Drive/Inputs/In/nState1 @bit 5 <-> STM Status/Status/Moving negative
//     Drive/Inputs/In/nState1 @bit 4 <-> STM Status/Status/Moving positive
//     Drive/Inputs/In/nState1 @bit 1 <-> STM Status/Status/Ready
//     Drive/Inputs/In/nState1 <-> STM Status/Status/Ready to enable
//     Drive/Inputs/In/nState1 @bit 6 <-> STM Status/Status/Torque reduced
//     Drive/Inputs/In/nState1 @bit 2 <-> STM Status/Status/Warning
//     Drive/Inputs/In/nState2 @bit 3 <-> STM Status/Status/Digital input 1
//     Drive/Inputs/In/nState2 @bit 4 <-> STM Status/Status/Digital input 2
//     Drive/Inputs/In/nState2 @bit 5 <-> STM Status/Status/Sync error
//     Drive/Inputs/In/nState2 @bit 7 <-> STM Status/Status/TxPDO Toggle
//     Drive/Inputs/In/nState4 @bit 1 <-> WcState/InputToggle
//     Drive/Inputs/In/nState4 <-> WcState/WcState
//     Drive/Outputs/Out/nCtrl1 <-> STM Control/Control/Enable
//     Drive/Outputs/Out/nCtrl1 @bit 2 <-> STM Control/Control/Reduce torque
//     Drive/Outputs/Out/nCtrl1 @bit 1 <-> STM Control/Control/Reset
//     Drive/Outputs/Out/nDataOut2[0] <-> STM Velocity/Velocity
//   (this object) <-> Device 1 (EtherCAT)/Term 1 (EK1200)/Term 5 (EK1122)/Box 6 (CU1124)/EK1100_M2L0/EL7041-1000_M2L0_Xdwn
//     Drive/Inputs/In/nState1 @bit 3 <-> STM Status/Status/Error
//     Drive/Inputs/In/nState1 @bit 5 <-> STM Status/Status/Moving negative
//     Drive/Inputs/In/nState1 @bit 4 <-> STM Status/Status/Moving positive
//     Drive/Inputs/In/nState1 @bit 1 <-> STM Status/Status/Ready
//     Drive/Inputs/In/nState1 <-> STM Status/Status/Ready to enable
//     Drive/Inputs/In/nState1 @bit 6 <-> STM Status/Status/Torque reduced
//     Drive/Inputs/In/nState1 @bit 2 <-> STM Status/Status/Warning
//     Drive/Inputs/In/nState2 @bit 3 <-> STM Status/Status/Digital input 1
//     Drive/Inputs/In/nState2 @bit 4 <-> STM Status/Status/Digital input 2
//     Drive/Inputs/In/nState2 @bit 5 <-> STM Status/Status/Sync error
//     Drive/Inputs/In/nState2 @bit 7 <-> STM Status/Status/TxPDO Toggle
//     Drive/Inputs/In/nState4 @bit 1 <-> WcState/InputToggle
//     Drive/Inputs/In/nState4 <-> WcState/WcState
//     Drive/Outputs/Out/nCtrl1 <-> STM Control/Control/Enable
//     Drive/Outputs/Out/nCtrl1 @bit 2 <-> STM Control/Control/Reduce torque
//     Drive/Outputs/Out/nCtrl1 @bit 1 <-> STM Control/Control/Reset
//     Drive/Outputs/Out/nDataOut2[0] <-> STM Velocity/Velocity
//   (this object) <-> Device 1 (EtherCAT)/Term 1 (EK1200)/Term 5 (EK1122)/Box 6 (CU1124)/EK1100_M2L0/EL5042_M2L0_PitchBender
//     Enc/Inputs/In/nComState @bit 1 <-> WcState/InputToggle
//     Enc/Inputs/In/nComState <-> WcState/WcState
//     Enc/Inputs/In/nDataIn1 <-> FB Inputs Channel 1/Position
//     Enc/Inputs/In/nDataIn1 <-> FB Inputs Channel 2/Position
//     Enc/Inputs/In/nState1 @bit 12 <-> FB Inputs Channel 1/Status/Diag
//     Enc/Inputs/In/nState1 @bit 12 <-> FB Inputs Channel 2/Status/Diag
//     Enc/Inputs/In/nState1 @bit 1 <-> FB Inputs Channel 1/Status/Error
//     Enc/Inputs/In/nState1 @bit 1 <-> FB Inputs Channel 2/Status/Error
//     Enc/Inputs/In/nState1 @bit 14 <-> FB Inputs Channel 1/Status/Input cycle counter
//     Enc/Inputs/In/nState1 @bit 14 <-> FB Inputs Channel 2/Status/Input cycle counter
//     Enc/Inputs/In/nState1 @bit 2 <-> FB Inputs Channel 1/Status/Ready
//     Enc/Inputs/In/nState1 @bit 2 <-> FB Inputs Channel 2/Status/Ready
//     Enc/Inputs/In/nState1 @bit 13 <-> FB Inputs Channel 1/Status/TxPDO State
//     Enc/Inputs/In/nState1 @bit 13 <-> FB Inputs Channel 2/Status/TxPDO State
//     Enc/Inputs/In/nState1 <-> FB Inputs Channel 1/Status/Warning
//     Enc/Inputs/In/nState1 <-> FB Inputs Channel 2/Status/Warning
//   (this object) <-> Device 1 (EtherCAT)/Term 1 (EK1200)/Term 5 (EK1122)/Box 6 (CU1124)/EK1100_M2L0/EL7041-1000_M2L0_PitchCoarse
//     Drive/Inputs/In/nState1 @bit 3 <-> STM Status/Status/Error
//     Drive/Inputs/In/nState1 @bit 5 <-> STM Status/Status/Moving negative
//     Drive/Inputs/In/nState1 @bit 4 <-> STM Status/Status/Moving positive
//     Drive/Inputs/In/nState1 @bit 1 <-> STM Status/Status/Ready
//     Drive/Inputs/In/nState1 <-> STM Status/Status/Ready to enable
//     Drive/Inputs/In/nState1 @bit 6 <-> STM Status/Status/Torque reduced
//     Drive/Inputs/In/nState1 @bit 2 <-> STM Status/Status/Warning
//     Drive/Inputs/In/nState2 @bit 3 <-> STM Status/Status/Digital input 1
//     Drive/Inputs/In/nState2 @bit 4 <-> STM Status/Status/Digital input 2
//     Drive/Inputs/In/nState2 @bit 5 <-> STM Status/Status/Sync error
//     Drive/Inputs/In/nState2 @bit 7 <-> STM Status/Status/TxPDO Toggle
//     Drive/Inputs/In/nState4 @bit 1 <-> WcState/InputToggle
//     Drive/Inputs/In/nState4 <-> WcState/WcState
//     Drive/Outputs/Out/nCtrl1 <-> STM Control/Control/Enable
//     Drive/Outputs/Out/nCtrl1 @bit 2 <-> STM Control/Control/Reduce torque
//     Drive/Outputs/Out/nCtrl1 @bit 1 <-> STM Control/Control/Reset
//     Drive/Outputs/Out/nDataOut2[0] <-> STM Velocity/Velocity
//   (this object) <-> Device 1 (EtherCAT)/Term 1 (EK1200)/Term 5 (EK1122)/Box 6 (CU1124)/EK1100_M2L0/EL7041-1000_M2L0_Bender
//     Drive/Inputs/In/nState1 @bit 3 <-> STM Status/Status/Error
//     Drive/Inputs/In/nState1 @bit 5 <-> STM Status/Status/Moving negative
//     Drive/Inputs/In/nState1 @bit 4 <-> STM Status/Status/Moving positive
//     Drive/Inputs/In/nState1 @bit 1 <-> STM Status/Status/Ready
//     Drive/Inputs/In/nState1 <-> STM Status/Status/Ready to enable
//     Drive/Inputs/In/nState1 @bit 6 <-> STM Status/Status/Torque reduced
//     Drive/Inputs/In/nState1 @bit 2 <-> STM Status/Status/Warning
//     Drive/Inputs/In/nState2 @bit 3 <-> STM Status/Status/Digital input 1
//     Drive/Inputs/In/nState2 @bit 4 <-> STM Status/Status/Digital input 2
//     Drive/Inputs/In/nState2 @bit 5 <-> STM Status/Status/Sync error
//     Drive/Inputs/In/nState2 @bit 7 <-> STM Status/Status/TxPDO Toggle
//     Drive/Inputs/In/nState4 @bit 1 <-> WcState/InputToggle
//     Drive/Inputs/In/nState4 <-> WcState/WcState
//     Drive/Outputs/Out/nCtrl1 <-> STM Control/Control/Enable
//     Drive/Outputs/Out/nCtrl1 @bit 2 <-> STM Control/Control/Reduce torque
//     Drive/Outputs/Out/nCtrl1 @bit 1 <-> STM Control/Control/Reset
//     Drive/Outputs/Out/nDataOut2[0] <-> STM Velocity/Velocity
//   (this object) <-> Device 1 (EtherCAT)/Term 1 (EK1200)/Term 5 (EK1122)/Box 6 (CU1124)/EK1100_SP1L0/EL5042_SP1L0_th1_th2
//     Enc/Inputs/In/nComState @bit 1 <-> WcState/InputToggle
//     Enc/Inputs/In/nComState <-> WcState/WcState
//     Enc/Inputs/In/nDataIn1 <-> FB Inputs Channel 1/Position
//     Enc/Inputs/In/nDataIn1 <-> FB Inputs Channel 2/Position
//     Enc/Inputs/In/nState1 @bit 12 <-> FB Inputs Channel 1/Status/Diag
//     Enc/Inputs/In/nState1 @bit 12 <-> FB Inputs Channel 2/Status/Diag
//     Enc/Inputs/In/nState1 @bit 1 <-> FB Inputs Channel 1/Status/Error
//     Enc/Inputs/In/nState1 @bit 1 <-> FB Inputs Channel 2/Status/Error
//     Enc/Inputs/In/nState1 @bit 14 <-> FB Inputs Channel 1/Status/Input cycle counter
//     Enc/Inputs/In/nState1 @bit 14 <-> FB Inputs Channel 2/Status/Input cycle counter
//     Enc/Inputs/In/nState1 @bit 2 <-> FB Inputs Channel 1/Status/Ready
//     Enc/Inputs/In/nState1 @bit 2 <-> FB Inputs Channel 2/Status/Ready
//     Enc/Inputs/In/nState1 @bit 13 <-> FB Inputs Channel 1/Status/TxPDO State
//     Enc/Inputs/In/nState1 @bit 13 <-> FB Inputs Channel 2/Status/TxPDO State
//     Enc/Inputs/In/nState1 <-> FB Inputs Channel 1/Status/Warning
//     Enc/Inputs/In/nState1 <-> FB Inputs Channel 2/Status/Warning
//   (this object) <-> Device 1 (EtherCAT)/Term 1 (EK1200)/Term 5 (EK1122)/Box 6 (CU1124)/EK1100_SP1L0/EL7047_SP1L0_th1
//     Drive/Inputs/In/nState1 @bit 3 <-> STM Status/Status/Error
//     Drive/Inputs/In/nState1 @bit 7 <-> STM Status/Status/Motor stall
//     Drive/Inputs/In/nState1 @bit 5 <-> STM Status/Status/Moving negative
//     Drive/Inputs/In/nState1 @bit 4 <-> STM Status/Status/Moving positive
//     Drive/Inputs/In/nState1 @bit 1 <-> STM Status/Status/Ready
//     Drive/Inputs/In/nState1 <-> STM Status/Status/Ready to enable
//     Drive/Inputs/In/nState1 @bit 6 <-> STM Status/Status/Torque reduced
//     Drive/Inputs/In/nState1 @bit 2 <-> STM Status/Status/Warning
//     Drive/Inputs/In/nState2 @bit 3 <-> STM Status/Status/Digital input 1
//     Drive/Inputs/In/nState2 @bit 4 <-> STM Status/Status/Digital input 2
//     Drive/Inputs/In/nState2 @bit 5 <-> STM Status/Status/Sync error
//     Drive/Inputs/In/nState2 @bit 7 <-> STM Status/Status/TxPDO Toggle
//     Drive/Inputs/In/nState4 @bit 1 <-> WcState/InputToggle
//     Drive/Inputs/In/nState4 <-> WcState/WcState
//     Drive/Outputs/Out/nCtrl1 <-> STM Control/Control/Enable
//     Drive/Outputs/Out/nCtrl1 @bit 2 <-> STM Control/Control/Reduce torque
//     Drive/Outputs/Out/nCtrl1 @bit 1 <-> STM Control/Control/Reset
//     Drive/Outputs/Out/nCtrl2 @bit 3 <-> STM Control/Control/Digital output 1
//     Drive/Outputs/Out/nDataOut2[0] <-> STM Velocity/Velocity
//   (this object) <-> Device 1 (EtherCAT)/Term 1 (EK1200)/Term 5 (EK1122)/Box 6 (CU1124)/EK1100_SP1L0/EL7047_SP1L0_th2
//     Drive/Inputs/In/nState1 @bit 3 <-> STM Status/Status/Error
//     Drive/Inputs/In/nState1 @bit 7 <-> STM Status/Status/Motor stall
//     Drive/Inputs/In/nState1 @bit 5 <-> STM Status/Status/Moving negative
//     Drive/Inputs/In/nState1 @bit 4 <-> STM Status/Status/Moving positive
//     Drive/Inputs/In/nState1 @bit 1 <-> STM Status/Status/Ready
//     Drive/Inputs/In/nState1 <-> STM Status/Status/Ready to enable
//     Drive/Inputs/In/nState1 @bit 6 <-> STM Status/Status/Torque reduced
//     Drive/Inputs/In/nState1 @bit 2 <-> STM Status/Status/Warning
//     Drive/Inputs/In/nState2 @bit 3 <-> STM Status/Status/Digital input 1
//     Drive/Inputs/In/nState2 @bit 4 <-> STM Status/Status/Digital input 2
//     Drive/Inputs/In/nState2 @bit 5 <-> STM Status/Status/Sync error
//     Drive/Inputs/In/nState2 @bit 7 <-> STM Status/Status/TxPDO Toggle
//     Drive/Inputs/In/nState4 @bit 1 <-> WcState/InputToggle
//     Drive/Inputs/In/nState4 <-> WcState/WcState
//     Drive/Outputs/Out/nCtrl1 <-> STM Control/Control/Enable
//     Drive/Outputs/Out/nCtrl1 @bit 2 <-> STM Control/Control/Reduce torque
//     Drive/Outputs/Out/nCtrl1 @bit 1 <-> STM Control/Control/Reset
//     Drive/Outputs/Out/nCtrl2 @bit 3 <-> STM Control/Control/Digital output 1
//     Drive/Outputs/Out/nDataOut2[0] <-> STM Velocity/Velocity
//   (this object) <-> Device 1 (EtherCAT)/Term 1 (EK1200)/Term 5 (EK1122)/Box 6 (CU1124)/EK1100_SP1L0/EL5042_SP1L0_tx_txd
//     Enc/Inputs/In/nComState @bit 1 <-> WcState/InputToggle
//     Enc/Inputs/In/nComState <-> WcState/WcState
//     Enc/Inputs/In/nDataIn1 <-> FB Inputs Channel 1/Position
//     Enc/Inputs/In/nDataIn1 <-> FB Inputs Channel 2/Position
//     Enc/Inputs/In/nState1 @bit 12 <-> FB Inputs Channel 1/Status/Diag
//     Enc/Inputs/In/nState1 @bit 12 <-> FB Inputs Channel 2/Status/Diag
//     Enc/Inputs/In/nState1 @bit 1 <-> FB Inputs Channel 1/Status/Error
//     Enc/Inputs/In/nState1 @bit 1 <-> FB Inputs Channel 2/Status/Error
//     Enc/Inputs/In/nState1 @bit 14 <-> FB Inputs Channel 1/Status/Input cycle counter
//     Enc/Inputs/In/nState1 @bit 14 <-> FB Inputs Channel 2/Status/Input cycle counter
//     Enc/Inputs/In/nState1 @bit 2 <-> FB Inputs Channel 1/Status/Ready
//     Enc/Inputs/In/nState1 @bit 2 <-> FB Inputs Channel 2/Status/Ready
//     Enc/Inputs/In/nState1 @bit 13 <-> FB Inputs Channel 1/Status/TxPDO State
//     Enc/Inputs/In/nState1 @bit 13 <-> FB Inputs Channel 2/Status/TxPDO State
//     Enc/Inputs/In/nState1 <-> FB Inputs Channel 1/Status/Warning
//     Enc/Inputs/In/nState1 <-> FB Inputs Channel 2/Status/Warning
//   (this object) <-> Device 1 (EtherCAT)/Term 1 (EK1200)/Term 5 (EK1122)/Box 6 (CU1124)/EK1100_SP1L0/EL7047_SP1L0_tx
//     Drive/Inputs/In/nState1 @bit 3 <-> STM Status/Status/Error
//     Drive/Inputs/In/nState1 @bit 7 <-> STM Status/Status/Motor stall
//     Drive/Inputs/In/nState1 @bit 5 <-> STM Status/Status/Moving negative
//     Drive/Inputs/In/nState1 @bit 4 <-> STM Status/Status/Moving positive
//     Drive/Inputs/In/nState1 @bit 1 <-> STM Status/Status/Ready
//     Drive/Inputs/In/nState1 <-> STM Status/Status/Ready to enable
//     Drive/Inputs/In/nState1 @bit 6 <-> STM Status/Status/Torque reduced
//     Drive/Inputs/In/nState1 @bit 2 <-> STM Status/Status/Warning
//     Drive/Inputs/In/nState2 @bit 3 <-> STM Status/Status/Digital input 1
//     Drive/Inputs/In/nState2 @bit 4 <-> STM Status/Status/Digital input 2
//     Drive/Inputs/In/nState2 @bit 5 <-> STM Status/Status/Sync error
//     Drive/Inputs/In/nState2 @bit 7 <-> STM Status/Status/TxPDO Toggle
//     Drive/Inputs/In/nState4 @bit 1 <-> WcState/InputToggle
//     Drive/Inputs/In/nState4 <-> WcState/WcState
//     Drive/Outputs/Out/nCtrl1 <-> STM Control/Control/Enable
//     Drive/Outputs/Out/nCtrl1 @bit 2 <-> STM Control/Control/Reduce torque
//     Drive/Outputs/Out/nCtrl1 @bit 1 <-> STM Control/Control/Reset
//     Drive/Outputs/Out/nCtrl2 @bit 3 <-> STM Control/Control/Digital output 1
//     Drive/Outputs/Out/nDataOut2[0] <-> STM Velocity/Velocity
//   (this object) <-> Device 1 (EtherCAT)/Term 1 (EK1200)/Term 5 (EK1122)/Box 6 (CU1124)/EK1100_SP1L0/EL7047_SP1L0_txd
//     Drive/Inputs/In/nState1 @bit 3 <-> STM Status/Status/Error
//     Drive/Inputs/In/nState1 @bit 7 <-> STM Status/Status/Motor stall
//     Drive/Inputs/In/nState1 @bit 5 <-> STM Status/Status/Moving negative
//     Drive/Inputs/In/nState1 @bit 4 <-> STM Status/Status/Moving positive
//     Drive/Inputs/In/nState1 @bit 1 <-> STM Status/Status/Ready
//     Drive/Inputs/In/nState1 <-> STM Status/Status/Ready to enable
//     Drive/Inputs/In/nState1 @bit 6 <-> STM Status/Status/Torque reduced
//     Drive/Inputs/In/nState1 @bit 2 <-> STM Status/Status/Warning
//     Drive/Inputs/In/nState2 @bit 3 <-> STM Status/Status/Digital input 1
//     Drive/Inputs/In/nState2 @bit 4 <-> STM Status/Status/Digital input 2
//     Drive/Inputs/In/nState2 @bit 5 <-> STM Status/Status/Sync error
//     Drive/Inputs/In/nState2 @bit 7 <-> STM Status/Status/TxPDO Toggle
//     Drive/Inputs/In/nState4 @bit 1 <-> WcState/InputToggle
//     Drive/Inputs/In/nState4 <-> WcState/WcState
//     Drive/Outputs/Out/nCtrl1 <-> STM Control/Control/Enable
//     Drive/Outputs/Out/nCtrl1 @bit 2 <-> STM Control/Control/Reduce torque
//     Drive/Outputs/Out/nCtrl1 @bit 1 <-> STM Control/Control/Reset
//     Drive/Outputs/Out/nCtrl2 @bit 3 <-> STM Control/Control/Digital output 1
//     Drive/Outputs/Out/nDataOut2[0] <-> STM Velocity/Velocity
//   (this object) <-> Device 1 (EtherCAT)/Term 1 (EK1200)/Term 5 (EK1122)/Box 6 (CU1124)/EK1100_SP1L0/EL5042_SP1L0_tyd
//     Enc/Inputs/In/nComState @bit 1 <-> WcState/InputToggle
//     Enc/Inputs/In/nComState <-> WcState/WcState
//     Enc/Inputs/In/nDataIn1 <-> FB Inputs Channel 1/Position
//     Enc/Inputs/In/nState1 @bit 12 <-> FB Inputs Channel 1/Status/Diag
//     Enc/Inputs/In/nState1 @bit 1 <-> FB Inputs Channel 1/Status/Error
//     Enc/Inputs/In/nState1 @bit 14 <-> FB Inputs Channel 1/Status/Input cycle counter
//     Enc/Inputs/In/nState1 @bit 2 <-> FB Inputs Channel 1/Status/Ready
//     Enc/Inputs/In/nState1 @bit 13 <-> FB Inputs Channel 1/Status/TxPDO State
//     Enc/Inputs/In/nState1 <-> FB Inputs Channel 1/Status/Warning
//   (this object) <-> Device 1 (EtherCAT)/Term 1 (EK1200)/Term 5 (EK1122)/Box 6 (CU1124)/EK1100_SP1L0/EL7047_SP1L0_tyd
//     Drive/Inputs/In/nState1 @bit 3 <-> STM Status/Status/Error
//     Drive/Inputs/In/nState1 @bit 7 <-> STM Status/Status/Motor stall
//     Drive/Inputs/In/nState1 @bit 5 <-> STM Status/Status/Moving negative
//     Drive/Inputs/In/nState1 @bit 4 <-> STM Status/Status/Moving positive
//     Drive/Inputs/In/nState1 @bit 1 <-> STM Status/Status/Ready
//     Drive/Inputs/In/nState1 <-> STM Status/Status/Ready to enable
//     Drive/Inputs/In/nState1 @bit 6 <-> STM Status/Status/Torque reduced
//     Drive/Inputs/In/nState1 @bit 2 <-> STM Status/Status/Warning
//     Drive/Inputs/In/nState2 @bit 3 <-> STM Status/Status/Digital input 1
//     Drive/Inputs/In/nState2 @bit 4 <-> STM Status/Status/Digital input 2
//     Drive/Inputs/In/nState2 @bit 5 <-> STM Status/Status/Sync error
//     Drive/Inputs/In/nState2 @bit 7 <-> STM Status/Status/TxPDO Toggle
//     Drive/Inputs/In/nState4 @bit 1 <-> WcState/InputToggle
//     Drive/Inputs/In/nState4 <-> WcState/WcState
//     Drive/Outputs/Out/nCtrl1 <-> STM Control/Control/Enable
//     Drive/Outputs/Out/nCtrl1 @bit 2 <-> STM Control/Control/Reduce torque
//     Drive/Outputs/Out/nCtrl1 @bit 1 <-> STM Control/Control/Reset
//     Drive/Outputs/Out/nCtrl2 @bit 3 <-> STM Control/Control/Digital output 1
//     Drive/Outputs/Out/nDataOut2[0] <-> STM Velocity/Velocity
//   lfe_optics Instance <-> Device 1 (EtherCAT)/Term 1 (EK1200)/PMPS_FFO
//     PlcTask Outputs/GVL_PMPS.g_FastFaultOutput1.q_xFastFaultOut <-> Channel 1/Output
//     PlcTask Outputs/GVL_PMPS.g_FastFaultOutput2.q_xFastFaultOut <-> Channel 2/Output
//   lfe_optics Instance <-> Device 1 (EtherCAT)/Term 1 (EK1200)/PMPS_PRE
//     PlcTask Inputs/PRG_PMPS.fbArbiterIO.i_stCurrentBP <-> IO Inputs/CurrentBP
//     PlcTask Inputs/PRG_PMPS.fbArbiterIO.xTxPDO_state <-> SYNC Inputs/TxPDO state
//     PlcTask Inputs/PRG_PMPS.fbArbiterIO.xTxPDO_toggle <-> SYNC Inputs/TxPDO toggle
//     PlcTask Outputs/PRG_PMPS.fbArbiterIO.q_stRequestedBP <-> IO Outputs/RequestedBP
//     PlcTask Outputs/PRG_PMPS.nMR1L0_Pitch_ENC_PMPS <-> IO Outputs/MR1L0_Pitch_ENC
//   lfe_optics Instance <-> Device 1 (EtherCAT)/Term 1 (EK1200)/Term 5 (EK1122)/Box 6 (CU1124)/EK1100_M2L0/EL1004_M2L0_STO
//     PlcTask Inputs/Main.M2L0.fbRunHOMS.bSTOEnable1 <-> Channel 1/Input
//     PlcTask Inputs/Main.M2L0.fbRunHOMS.bSTOEnable2 <-> Channel 2/Input
//   lfe_optics Instance <-> Device 1 (EtherCAT)/Term 1 (EK1200)/Term 5 (EK1122)/Box 6 (CU1124)/EK1100_M2L0/EL3054_M2L0_FWM_PRSM
//     PlcTask Inputs/PRG_MR2L0_HOMS.fbCoolingPanel.fbFlow_1.iRaw <-> AI Standard Channel 1/Value
//     PlcTask Inputs/PRG_MR2L0_HOMS.fbCoolingPanel.fbFlow_2.iRaw <-> AI Standard Channel 2/Value
//     PlcTask Inputs/PRG_MR2L0_HOMS.fbCoolingPanel.fbPress_1.iRaw <-> AI Standard Channel 3/Value
//   lfe_optics Instance <-> Device 1 (EtherCAT)/Term 1 (EK1200)/Term 5 (EK1122)/Box 6 (CU1124)/EK1100_M2L0/EL5042_M2L0_PitchBender
//     PlcTask Inputs/GVL_M2L0.M2L0_Pitch.diEncCnt <-> FB Inputs Channel 1/Position
//     PlcTask Inputs/Main.M11.nRawEncoderULINT <-> FB Inputs Channel 1/Position
//     PlcTask Inputs/Main.M12.nRawEncoderULINT <-> FB Inputs Channel 2/Position
//   lfe_optics Instance <-> Device 1 (EtherCAT)/Term 1 (EK1200)/Term 5 (EK1122)/Box 6 (CU1124)/EK1100_M2L0/EL5042_M2L0_Xupdwn
//     PlcTask Inputs/Main.M2L0.fbRunHOMS.stXdwnEnc/Count <-> FB Inputs Channel 2/Position
//     PlcTask Inputs/Main.M2L0.fbRunHOMS.stXupEnc/Count <-> FB Inputs Channel 1/Position
//   lfe_optics Instance <-> Device 1 (EtherCAT)/Term 1 (EK1200)/Term 5 (EK1122)/Box 6 (CU1124)/EK1100_M2L0/EL5042_M2L0_Yupdwn
//     PlcTask Inputs/Main.M2L0.fbRunHOMS.stYdwnEnc/Count <-> FB Inputs Channel 2/Position
//     PlcTask Inputs/Main.M2L0.fbRunHOMS.stYupEnc/Count <-> FB Inputs Channel 1/Position
//     PlcTask Inputs/Main.M7.nRawEncoderULINT <-> FB Inputs Channel 1/Position
//   lfe_optics Instance <-> Device 1 (EtherCAT)/Term 1 (EK1200)/Term 5 (EK1122)/Box 6 (CU1124)/EK1100_M2L0/EL7041-1000_M2L0_Bender
//     PlcTask Inputs/Main.M12.bLimitBackwardEnable <-> STM Status/Status/Digital input 2
//     PlcTask Inputs/Main.M12.bLimitForwardEnable <-> STM Status/Status/Digital input 1
//   lfe_optics Instance <-> Device 1 (EtherCAT)/Term 1 (EK1200)/Term 5 (EK1122)/Box 6 (CU1124)/EK1100_M2L0/EL7041-1000_M2L0_PitchCoarse
//     PlcTask Inputs/Main.M11.bLimitBackwardEnable <-> STM Status/Status/Digital input 2
//     PlcTask Inputs/Main.M11.bLimitForwardEnable <-> STM Status/Status/Digital input 1
//   lfe_optics Instance <-> Device 1 (EtherCAT)/Term 1 (EK1200)/Term 5 (EK1122)/Box 6 (CU1124)/EK1100_M2L0/EL7041-1000_M2L0_Xdwn
//     PlcTask Inputs/Main.M10.bLimitBackwardEnable <-> STM Status/Status/Digital input 2
//     PlcTask Inputs/Main.M10.bLimitForwardEnable <-> STM Status/Status/Digital input 1
//   lfe_optics Instance <-> Device 1 (EtherCAT)/Term 1 (EK1200)/Term 5 (EK1122)/Box 6 (CU1124)/EK1100_M2L0/EL7041-1000_M2L0_Xup
//     PlcTask Inputs/Main.M9.bLimitBackwardEnable <-> STM Status/Status/Digital input 2
//     PlcTask Inputs/Main.M9.bLimitForwardEnable <-> STM Status/Status/Digital input 1
//   lfe_optics Instance <-> Device 1 (EtherCAT)/Term 1 (EK1200)/Term 5 (EK1122)/Box 6 (CU1124)/EK1100_M2L0/EL7041-1000_M2L0_Ydwn
//     PlcTask Inputs/Main.M8.bLimitBackwardEnable <-> STM Status/Status/Digital input 2
//     PlcTask Inputs/Main.M8.bLimitForwardEnable <-> STM Status/Status/Digital input 1
//   lfe_optics Instance <-> Device 1 (EtherCAT)/Term 1 (EK1200)/Term 5 (EK1122)/Box 6 (CU1124)/EK1100_M2L0/EL7041-1000_M2L0_Yup
//     PlcTask Inputs/Main.M7.bLimitBackwardEnable <-> STM Status/Status/Digital input 2
//     PlcTask Inputs/Main.M7.bLimitForwardEnable <-> STM Status/Status/Digital input 1
//   lfe_optics Instance <-> Device 1 (EtherCAT)/Term 1 (EK1200)/Term 5 (EK1122)/Box 6 (CU1124)/EK1100_SP1L0/EL1008_SP1L0_STO_DI
//     PlcTask Inputs/Main.bDI7 <-> Channel 8/Input
//     PlcTask Inputs/Main.bSTO <-> Channel 7/Input
//     PlcTask Inputs/Main.bTH1_NOTL <-> Channel 2/Input
//     PlcTask Inputs/Main.bTH2_NOTL <-> Channel 4/Input
//     PlcTask Inputs/Main.bTH1_POTL <-> Channel 1/Input
//     PlcTask Inputs/Main.bTH2_POTL <-> Channel 3/Input
//     PlcTask Inputs/Main.bTX_NOTL <-> Channel 6/Input
//     PlcTask Inputs/Main.bTX_POTL <-> Channel 5/Input
//   lfe_optics Instance <-> Device 1 (EtherCAT)/Term 1 (EK1200)/Term 5 (EK1122)/Box 6 (CU1124)/EK1100_SP1L0/EL2008_SP1L0_DO
//     PlcTask Outputs/Main.bDO{1..6} <-> Channel {2..7}/Output  (6 links)
//     PlcTask Outputs/Main.bFanOn <-> Channel 8/Output
//     PlcTask Outputs/Main.bTx_Brake_Solenoid <-> Channel 1/Output
//   lfe_optics Instance <-> Device 1 (EtherCAT)/Term 1 (EK1200)/Term 5 (EK1122)/Box 6 (CU1124)/EK1100_SP1L0/EL3054_SP1L0_AI
//     PlcTask Inputs/Main.nAI <-> AI Standard Channel 1/Value
//   lfe_optics Instance <-> Device 1 (EtherCAT)/Term 1 (EK1200)/Term 5 (EK1122)/Box 6 (CU1124)/EK1100_SP1L0/EL5042_SP1L0_th1_th2
//     PlcTask Inputs/Main.M13.nRawEncoderULINT <-> FB Inputs Channel 1/Position
//     PlcTask Inputs/Main.M14.nRawEncoderULINT <-> FB Inputs Channel 2/Position
//   lfe_optics Instance <-> Device 1 (EtherCAT)/Term 1 (EK1200)/Term 5 (EK1122)/Box 6 (CU1124)/EK1100_SP1L0/EL5042_SP1L0_tx_txd
//     PlcTask Inputs/Main.M15.nRawEncoderULINT <-> FB Inputs Channel 1/Position
//     PlcTask Inputs/Main.M16.nRawEncoderULINT <-> FB Inputs Channel 2/Position
//   lfe_optics Instance <-> Device 1 (EtherCAT)/Term 1 (EK1200)/Term 5 (EK1122)/Box 6 (CU1124)/EK1100_SP1L0/EL5042_SP1L0_tyd
//     PlcTask Inputs/Main.M17.nRawEncoderULINT <-> FB Inputs Channel 1/Position
//   lfe_optics Instance <-> Device 1 (EtherCAT)/Term 1 (EK1200)/Term 5 (EK1122)/Box 6 (CU1124)/EK1100_SP1L0/EL7047_SP1L0_th1
//     PlcTask Inputs/Main.M13.bLimitBackwardEnable <-> STM Status/Status/Digital input 2
//     PlcTask Inputs/Main.M13.bLimitForwardEnable <-> STM Status/Status/Digital input 1
//   lfe_optics Instance <-> Device 1 (EtherCAT)/Term 1 (EK1200)/Term 5 (EK1122)/Box 6 (CU1124)/EK1100_SP1L0/EL7047_SP1L0_th2
//     PlcTask Inputs/Main.M14.bLimitBackwardEnable <-> STM Status/Status/Digital input 2
//     PlcTask Inputs/Main.M14.bLimitForwardEnable <-> STM Status/Status/Digital input 1
//   lfe_optics Instance <-> Device 1 (EtherCAT)/Term 1 (EK1200)/Term 5 (EK1122)/Box 6 (CU1124)/EK1100_SP1L0/EL7047_SP1L0_tx
//     PlcTask Inputs/Main.M15.bLimitBackwardEnable <-> STM Status/Status/Digital input 2
//     PlcTask Inputs/Main.M15.bLimitForwardEnable <-> STM Status/Status/Digital input 1
//   lfe_optics Instance <-> Device 1 (EtherCAT)/Term 1 (EK1200)/Term 5 (EK1122)/Box 6 (CU1124)/EK1100_SP1L0/EL7047_SP1L0_txd
//     PlcTask Inputs/Main.M16.bLimitBackwardEnable <-> STM Status/Status/Digital input 2
//     PlcTask Inputs/Main.M16.bLimitForwardEnable <-> STM Status/Status/Digital input 1
//   lfe_optics Instance <-> Device 1 (EtherCAT)/Term 1 (EK1200)/Term 5 (EK1122)/Box 6 (CU1124)/EK1100_SP1L0/EL7047_SP1L0_tyd
//     PlcTask Inputs/Main.M17.bLimitBackwardEnable <-> STM Status/Status/Digital input 2
//     PlcTask Inputs/Main.M17.bLimitForwardEnable <-> STM Status/Status/Digital input 1
//   lfe_optics Instance <-> Device 1 (EtherCAT)/Term 1 (EK1200)/Term 5 (EK1122)/Box 6 (CU1124)/EP2008-0001_M1M2_VCV
//     PlcTask Outputs/PRG_MR1L0_HOMS.bActivateVarCoolMR1L0 <-> Channel 1/Output
//     PlcTask Outputs/PRG_MR2L0_HOMS.bActivateVarCoolMR2L0 <-> Channel 2/Output
//   lfe_optics Instance <-> Device 1 (EtherCAT)/Term 1 (EK1200)/Term 5 (EK1122)/EK1100_M1L0/EL1004_M1L0_STO
//     PlcTask Inputs/Main.M1L0.fbRunHOMS.bSTOEnable1 <-> Channel 1/Input
//     PlcTask Inputs/Main.M1L0.fbRunHOMS.bSTOEnable2 <-> Channel 2/Input
//   lfe_optics Instance <-> Device 1 (EtherCAT)/Term 1 (EK1200)/Term 5 (EK1122)/EK1100_M1L0/EL3054_M1L0_FWM_PRSM
//     PlcTask Inputs/PRG_MR1L0_HOMS.fbCoolingPanel.fbFlow_1.iRaw <-> AI Standard Channel 1/Value
//     PlcTask Inputs/PRG_MR1L0_HOMS.fbCoolingPanel.fbFlow_2.iRaw <-> AI Standard Channel 2/Value
//     PlcTask Inputs/PRG_MR1L0_HOMS.fbCoolingPanel.fbPress_1.iRaw <-> AI Standard Channel 3/Value
//   lfe_optics Instance <-> Device 1 (EtherCAT)/Term 1 (EK1200)/Term 5 (EK1122)/EK1100_M1L0/EL5042_M1L0_PitchBender
//     PlcTask Inputs/GVL_M1L0.M1L0_Pitch.diEncCnt <-> FB Inputs Channel 1/Position
//     PlcTask Inputs/Main.M5.nRawEncoderULINT <-> FB Inputs Channel 1/Position
//     PlcTask Inputs/Main.M6.nRawEncoderULINT <-> FB Inputs Channel 2/Position
//   lfe_optics Instance <-> Device 1 (EtherCAT)/Term 1 (EK1200)/Term 5 (EK1122)/EK1100_M1L0/EL5042_M1L0_Xupdwn
//     PlcTask Inputs/Main.M1L0.fbRunHOMS.stXdwnEnc/Count <-> FB Inputs Channel 2/Position
//     PlcTask Inputs/Main.M1L0.fbRunHOMS.stXupEnc/Count <-> FB Inputs Channel 1/Position
//     PlcTask Inputs/Main.M3.nRawEncoderULINT <-> FB Inputs Channel 1/Position
//     PlcTask Inputs/Main.M9.nRawEncoderULINT <-> FB Inputs Channel 1/Position
//   lfe_optics Instance <-> Device 1 (EtherCAT)/Term 1 (EK1200)/Term 5 (EK1122)/EK1100_M1L0/EL5042_M1L0_Yupdwn
//     PlcTask Inputs/Main.M1.nRawEncoderULINT <-> FB Inputs Channel 1/Position
//     PlcTask Inputs/Main.M1L0.fbRunHOMS.stYdwnEnc/Count <-> FB Inputs Channel 2/Position
//     PlcTask Inputs/Main.M1L0.fbRunHOMS.stYupEnc/Count <-> FB Inputs Channel 1/Position
//   lfe_optics Instance <-> Device 1 (EtherCAT)/Term 1 (EK1200)/Term 5 (EK1122)/EK1100_M1L0/EL6001_M1L0_PitchFine
//     SerialIO Inputs/GVL_SerialIO.Serial_stComIn_M1L0/D[{0..21}] <-> COM Inputs/Data In {0..21}  (22 links)
//     SerialIO Inputs/GVL_SerialIO.Serial_stComIn_M1L0/Status <-> COM Inputs/Status
//     SerialIO Outputs/GVL_SerialIO.Serial_stComOut_M1L0/Ctrl <-> COM Outputs/Ctrl
//     SerialIO Outputs/GVL_SerialIO.Serial_stComOut_M1L0/D[{0..21}] <-> COM Outputs/Data Out {0..21}  (22 links)
//   lfe_optics Instance <-> Device 1 (EtherCAT)/Term 1 (EK1200)/Term 5 (EK1122)/EK1100_M1L0/EL7041-1000_M1L0_Bender
//     PlcTask Inputs/Main.M6.bLimitBackwardEnable <-> STM Status/Status/Digital input 2
//     PlcTask Inputs/Main.M6.bLimitForwardEnable <-> STM Status/Status/Digital input 1
//   lfe_optics Instance <-> Device 1 (EtherCAT)/Term 1 (EK1200)/Term 5 (EK1122)/EK1100_M1L0/EL7041-1000_M1L0_PitchCoarse
//     PlcTask Inputs/Main.M5.bLimitBackwardEnable <-> STM Status/Status/Digital input 2
//     PlcTask Inputs/Main.M5.bLimitForwardEnable <-> STM Status/Status/Digital input 1
//   lfe_optics Instance <-> Device 1 (EtherCAT)/Term 1 (EK1200)/Term 5 (EK1122)/EK1100_M1L0/EL7041-1000_M1L0_Xdwn
//     PlcTask Inputs/Main.M4.bLimitBackwardEnable <-> STM Status/Status/Digital input 2
//     PlcTask Inputs/Main.M4.bLimitForwardEnable <-> STM Status/Status/Digital input 1
//   lfe_optics Instance <-> Device 1 (EtherCAT)/Term 1 (EK1200)/Term 5 (EK1122)/EK1100_M1L0/EL7041-1000_M1L0_Xup
//     PlcTask Inputs/Main.M3.bLimitBackwardEnable <-> STM Status/Status/Digital input 2
//     PlcTask Inputs/Main.M3.bLimitForwardEnable <-> STM Status/Status/Digital input 1
//   lfe_optics Instance <-> Device 1 (EtherCAT)/Term 1 (EK1200)/Term 5 (EK1122)/EK1100_M1L0/EL7041-1000_M1L0_Ydwn
//     PlcTask Inputs/Main.M2.bLimitBackwardEnable <-> STM Status/Status/Digital input 2
//     PlcTask Inputs/Main.M2.bLimitForwardEnable <-> STM Status/Status/Digital input 1
//   lfe_optics Instance <-> Device 1 (EtherCAT)/Term 1 (EK1200)/Term 5 (EK1122)/EK1100_M1L0/EL7041-1000_M1L0_Yup
//     PlcTask Inputs/Main.M1.bLimitBackwardEnable <-> STM Status/Status/Digital input 2
//     PlcTask Inputs/Main.M1.bLimitForwardEnable <-> STM Status/Status/Digital input 1
//   lfe_optics Instance <-> NC-Task 1 SAF/Axes/M1L0-Bender
//     PlcTask Inputs/Main.M6.Axis.NcToPlc <-> Outputs/ToPlc
//     PlcTask Outputs/Main.M6.Axis.PlcToNc <-> Inputs/FromPlc
//   lfe_optics Instance <-> NC-Task 1 SAF/Axes/M1L0-Pitch
//     PlcTask Inputs/Main.M5.Axis.NcToPlc <-> Outputs/ToPlc
//     PlcTask Outputs/Main.M5.Axis.PlcToNc <-> Inputs/FromPlc
//   lfe_optics Instance <-> NC-Task 1 SAF/Axes/M1L0-Xdwn
//     PlcTask Inputs/Main.M4.Axis.NcToPlc <-> Outputs/ToPlc
//     PlcTask Outputs/Main.M4.Axis.PlcToNc <-> Inputs/FromPlc
//   lfe_optics Instance <-> NC-Task 1 SAF/Axes/M1L0-Xup
//     PlcTask Inputs/Main.M3.Axis.NcToPlc <-> Outputs/ToPlc
//     PlcTask Outputs/Main.M3.Axis.PlcToNc <-> Inputs/FromPlc
//   lfe_optics Instance <-> NC-Task 1 SAF/Axes/M1L0-Ydwn
//     PlcTask Inputs/Main.M2.Axis.NcToPlc <-> Outputs/ToPlc
//     PlcTask Outputs/Main.M2.Axis.PlcToNc <-> Inputs/FromPlc
//   lfe_optics Instance <-> NC-Task 1 SAF/Axes/M1L0-Yup
//     PlcTask Inputs/Main.M1.Axis.NcToPlc <-> Outputs/ToPlc
//     PlcTask Outputs/Main.M1.Axis.PlcToNc <-> Inputs/FromPlc
//   lfe_optics Instance <-> NC-Task 1 SAF/Axes/M2L0-Bender
//     PlcTask Inputs/Main.M12.Axis.NcToPlc <-> Outputs/ToPlc
//     PlcTask Outputs/Main.M12.Axis.PlcToNc <-> Inputs/FromPlc
//   lfe_optics Instance <-> NC-Task 1 SAF/Axes/M2L0-Pitch
//     PlcTask Inputs/Main.M11.Axis.NcToPlc <-> Outputs/ToPlc
//     PlcTask Outputs/Main.M11.Axis.PlcToNc <-> Inputs/FromPlc
//   lfe_optics Instance <-> NC-Task 1 SAF/Axes/M2L0-Xdwn
//     PlcTask Inputs/Main.M10.Axis.NcToPlc <-> Outputs/ToPlc
//     PlcTask Outputs/Main.M10.Axis.PlcToNc <-> Inputs/FromPlc
//   lfe_optics Instance <-> NC-Task 1 SAF/Axes/M2L0-Xup
//     PlcTask Inputs/Main.M9.Axis.NcToPlc <-> Outputs/ToPlc
//     PlcTask Outputs/Main.M9.Axis.PlcToNc <-> Inputs/FromPlc
//   lfe_optics Instance <-> NC-Task 1 SAF/Axes/M2L0-Ydwn
//     PlcTask Inputs/Main.M8.Axis.NcToPlc <-> Outputs/ToPlc
//     PlcTask Outputs/Main.M8.Axis.PlcToNc <-> Inputs/FromPlc
//   lfe_optics Instance <-> NC-Task 1 SAF/Axes/M2L0-Yup
//     PlcTask Inputs/Main.M7.Axis.NcToPlc <-> Outputs/ToPlc
//     PlcTask Outputs/Main.M7.Axis.PlcToNc <-> Inputs/FromPlc
//   lfe_optics Instance <-> NC-Task 1 SAF/Axes/SP1L0-TH1
//     PlcTask Inputs/Main.M13.Axis.NcToPlc <-> Outputs/ToPlc
//     PlcTask Outputs/Main.M13.Axis.PlcToNc <-> Inputs/FromPlc
//   lfe_optics Instance <-> NC-Task 1 SAF/Axes/SP1L0-TH2
//     PlcTask Inputs/Main.M14.Axis.NcToPlc <-> Outputs/ToPlc
//     PlcTask Outputs/Main.M14.Axis.PlcToNc <-> Inputs/FromPlc
//   lfe_optics Instance <-> NC-Task 1 SAF/Axes/SP1L0-Tx
//     PlcTask Inputs/Main.M15.Axis.NcToPlc <-> Outputs/ToPlc
//     PlcTask Outputs/Main.M15.Axis.PlcToNc <-> Inputs/FromPlc
//   lfe_optics Instance <-> NC-Task 1 SAF/Axes/SP1L0-Txd
//     PlcTask Inputs/Main.M16.Axis.NcToPlc <-> Outputs/ToPlc
//     PlcTask Outputs/Main.M16.Axis.PlcToNc <-> Inputs/FromPlc
//   lfe_optics Instance <-> NC-Task 1 SAF/Axes/SP1L0-Tyd
//     PlcTask Inputs/Main.M17.Axis.NcToPlc <-> Outputs/ToPlc
//     PlcTask Outputs/Main.M17.Axis.PlcToNc <-> Inputs/FromPlc

CONFIGURATION lfe_optics
    RESOURCE PLC ON TwinCAT3
        TASK PiezoDriver(INTERVAL := T#1ms, PRIORITY := 3);
        TASK PlcTask(INTERVAL := T#10ms, PRIORITY := 20);
        PROGRAM PiezoSerial WITH PiezoDriver : PiezoSerial;
        PROGRAM Main WITH PlcTask : Main;
        PROGRAM PRG_1_PlcTask WITH PlcTask : PRG_1_PlcTask;
    END_RESOURCE
END_CONFIGURATION

// ---- DUTs/E_MR1L0_CoatingStates.TcDUT
{attribute 'qualified_only'}
{attribute 'strict'}
TYPE E_MR1L0_CoatingStates :
(
    Unknown := 0,
    L0B4C := 1,
    L0Ni := 2,
    L1B4C := 3,
    L1Ni := 4
) UINT;
END_TYPE

// ---- DUTs/E_MR2L0_CoatingStates.TcDUT
{attribute 'qualified_only'}
{attribute 'strict'}
TYPE E_MR2L0_CoatingStates :
(
    Unknown := 0,
    B4C := 1,
    Ni := 2
) UINT;
END_TYPE

// ---- Version/Global_Version.TcGVL
{attribute 'TcGenerated'}
{attribute 'no-analysis'}
{attribute 'linkalways'}
// This function has been automatically generated from the project information.
VAR_GLOBAL CONSTANT
    {attribute 'const_non_replaced'}
    stLibVersion_lcls_plc_lfe_optics : ST_LibVersion := (iMajor := 4, iMinor := 0, iBuild := 0, iRevision := 0, nFlags := 1, sVersion := '4.0.0');
END_VAR

// ---- GVLs/GVL_COM_Buffers.TcGVL
VAR_GLOBAL
    // M1L0
    Serial_RXBuffer_M1L0 : ComBuffer;
    Serial_TXBuffer_M1L0 : ComBuffer;

    // M2L0
    Serial_RXBuffer_M2L0 : ComBuffer;
    Serial_TXBuffer_M2L0 : ComBuffer;
END_VAR

// ---- GVLs/GVL_M1L0.TcGVL
{attribute 'qualified_only'}
VAR_GLOBAL
    // Pitch Mechanism:
    {attribute 'TcLinkTo' := '.diEncCnt:=TIIB[EL5042_M1L0_PitchBender]^FB Inputs Channel 1^Position'}
    M1L0_Pitch : HOMS_PitchMechanism := (ReqPosLimHi := 120.0,
                                         ReqPosLimLo := -182.0,
                                         diEncPosLimHi := 8662020,
                                         diEncPosLimLo := 8507095);
END_VAR

// ---- GVLs/GVL_M1L0_Constants.TcGVL
{attribute 'qualified_only'}
VAR_GLOBAL CONSTANT
    // Encoder reference values in counts = nm
    // Enc Ref Vals from alignment 2020-5-27
    nYUP_ENC_REF : ULINT := 16171800;
    nYDWN_ENC_REF : ULINT := 14866900;
    nXUP_ENC_REF : ULINT := 24901730;
    nXDWN_ENC_REF : ULINT := 22921460;
END_VAR

// ---- GVLs/GVL_M2L0.TcGVL
{attribute 'qualified_only'}
VAR_GLOBAL
    // Pitch Mechanism
    {attribute 'TcLinkTo' := '.diEncCnt:=TIIB[EL5042_M2L0_PitchBender]^FB Inputs Channel 1^Position'}
    M2L0_Pitch : HOMS_PitchMechanism := (ReqPosLimHi := 154.9,
                                         ReqPosLimLo := -45.1,
                                         diEncPosLimHi := 9550777,
                                         diEncPosLimLo := 9448178);
END_VAR

// ---- GVLs/GVL_M2L0_Constants.TcGVL
{attribute 'qualified_only'}
VAR_GLOBAL CONSTANT
    // Encoder reference values in counts = nm
    // Encoder reference values after alignment 5-29-20
    nYUP_ENC_REF : ULINT := 12018200;
    nYDWN_ENC_REF : ULINT := 15143700;
    nXUP_ENC_REF : ULINT := 25363400;
    nXDWN_ENC_REF : ULINT := 24398100;
END_VAR

// ---- GVLs/GVL_PMPS.TcGVL
{attribute 'qualified_only'}
VAR_GLOBAL
    // Implementation of the FFO
    {attribute 'pytmc' := '
        pv: PLC:LFE:OPTICS:FFO:01
    '}
    {attribute 'TcLinkTo' := '.q_xFastFaultOut:=TIIB[PMPS_FFO]^Channel 1^Output'}
    g_FastFaultOutput1 : FB_HardwareFFOutput := (bAutoReset:=TRUE, i_sNetID:='172.21.88.66.1.1');

    {attribute 'pytmc' := '
        pv: PLC:LFE:OPTICS:FFO:02
    '}
    {attribute 'TcLinkTo' := '.q_xFastFaultOut:=TIIB[PMPS_FFO]^Channel 2^Output'}
    g_FastFaultOutput2 : FB_HardwareFFOutput := (bAutoReset:=TRUE, i_sNetID:='172.21.88.66.1.1');

    {attribute 'pytmc' := '
        pv: PLC:LFE:OPTICS:ARB:01
    '}
    g_fbArbiter1 : FB_Arbiter(1);

    {attribute 'pytmc' := '
        pv: PLC:LFE:OPTICS:ARB:02
    '}
    g_fbArbiter2 : FB_Arbiter(2);
END_VAR

// ---- GVLs/GVL_SerialIO.TcGVL
VAR_GLOBAL
    //Better have your inputs and outputs!
    // M1L0
    Serial_stComIn_M1L0 AT %I* : EL6inData22B; // M1L0 In Serial Comm Array
    Serial_stComOut_M1L0 AT %Q* : EL6outData22B; // M1L0 Out Serual Comm Array

    // M2L0
    Serial_stComIn_M2L0 AT %I* : EL6inData22B; // M2L0 In Serial Comm Array
    Serial_stComOut_M2L0 AT %Q* : EL6outData22B; // M2L0 Out Serial Comm Array
END_VAR

// ---- GVLs/GVL_States.TcGVL
{attribute 'qualified_only'}
VAR_GLOBAL
    stDefaultY : ST_PositionState := (
        fDelta:=100,
        fVelocity:=100,
        fAccel:=200,
        fDecel:=200,
        bMoveOk:=TRUE,
        bValid:=TRUE,
        bUseRawCounts:=TRUE
    );
END_VAR

// ---- POUs/Serial Comm/PiezoSerial.TcPOU
PROGRAM PiezoSerial
VAR
    //PI Serial
    fbE621SerialDriver_M1L0 : FB_PI_E621_SerialDriver;
    rtInitParams_M1L0	:	R_TRIG;
    tonTimeoutRst_M1L0	: TON := (PT:=T#2S); //For timeout reset

    fbE621SerialDriver_M2L0 : FB_PI_E621_SerialDriver;
    rtInitParams_M2L0	:	R_TRIG;
    tonTimeoutRst_M2L0	: TON := (PT:=T#2S); //For timeout reset
END_VAR

//Piezo E-621
///////////////////////
fbE621SerialDriver_M1L0.i_xExecute := TRUE;
fbE621SerialDriver_M1L0.i_xExecute R= fbE621SerialDriver_M1L0.q_xDone;
fbE621SerialDriver_M1L0(iq_stPiezoAxis:= GVL_M1L0.M1L0_Pitch.Piezo,
                        iq_stSerialRXBuffer:= Serial_RXBuffer_M1L0,
                        iq_stSerialTXBuffer:= Serial_TXBuffer_M1L0);

fbE621SerialDriver_M2L0.i_xExecute := TRUE;
fbE621SerialDriver_M2L0.i_xExecute R= fbE621SerialDriver_M2L0.q_xDone;
fbE621SerialDriver_M2L0(iq_stPiezoAxis:= GVL_M2L0.M2L0_Pitch.Piezo,
                        iq_stSerialRXBuffer:= Serial_RXBuffer_M2L0,
                        iq_stSerialTXBuffer:= Serial_TXBuffer_M2L0);

END_PROGRAM

// ---- POUs/Main.TcPOU
PROGRAM Main
VAR
    // M1L0
    // Motors
    {attribute 'TcLinkTo' := '.bLimitForwardEnable:=TIIB[EL7041-1000_M1L0_Yup]^STM Status^Status^Digital input 1;
                              .bLimitBackwardEnable:=TIIB[EL7041-1000_M1L0_Yup]^STM Status^Status^Digital input 2;
                              .nRawEncoderULINT:=TIIB[EL5042_M1L0_Yupdwn]^FB Inputs Channel 1^Position'}
    {attribute 'pytmc' := '
        pv: MR1L0:HOMS:MMS:YUP
    '}
    M1 : ST_MotionStage := (fVelocity:=200.0, nEnableMode:=ENUM_StageEnableMode.ALWAYS, bPowerSelf:=TRUE, sName:='MR1L0_YUP'); // M1L0 Yup
    fbMotionStage_m1 : FB_MotionStage;

    {attribute 'TcLinkTo' := '.bLimitForwardEnable:=TIIB[EL7041-1000_M1L0_Ydwn]^STM Status^Status^Digital input 1;
                              .bLimitBackwardEnable:=TIIB[EL7041-1000_M1L0_Ydwn]^STM Status^Status^Digital input 2'}
    {attribute 'pytmc' := '
        pv: MR1L0:HOMS:MMS:YDWN
    '}
    M2 : ST_MotionStage := (fVelocity:=200.0, nEnableMode:=ENUM_StageEnableMode.ALWAYS, bPowerSelf:=TRUE, sName:='MR1L0_YDWN'); // M1L0 Ydwn
    fbMotionStage_m2 : FB_MotionStage;

    {attribute 'TcLinkTo' := '.bLimitForwardEnable:=TIIB[EL7041-1000_M1L0_Xup]^STM Status^Status^Digital input 1;
                              .bLimitBackwardEnable:=TIIB[EL7041-1000_M1L0_Xup]^STM Status^Status^Digital input 2;
                              .nRawEncoderULINT:=TIIB[EL5042_M1L0_Xupdwn]^FB Inputs Channel 1^Position'}
    {attribute 'pytmc' := '
        pv: MR1L0:HOMS:MMS:XUP
    '}
    M3 : ST_MotionStage := (fVelocity:=1000.0, nEnableMode:=ENUM_StageEnableMode.ALWAYS, bPowerSelf:=TRUE, sName:='MR1L0_XUP'); // M1L0 Xup
    fbMotionStage_m3 : FB_MotionStage;

    {attribute 'TcLinkTo' := '.bLimitForwardEnable:=TIIB[EL7041-1000_M1L0_Xdwn]^STM Status^Status^Digital input 1;
                              .bLimitBackwardEnable:=TIIB[EL7041-1000_M1L0_Xdwn]^STM Status^Status^Digital input 2'}
    {attribute 'pytmc' := '
        pv: MR1L0:HOMS:MMS:XDWN
    '}
    M4 : ST_MotionStage := (fVelocity:=1000.0, nEnableMode:=ENUM_StageEnableMode.ALWAYS, bPowerSelf:=TRUE, sName:='MR1L0_XDWN'); // M1L0 Xdwn
    fbMotionStage_m4 : FB_MotionStage;

    {attribute 'TcLinkTo' := '.bLimitForwardEnable:=TIIB[EL7041-1000_M1L0_PitchCoarse]^STM Status^Status^Digital input 1;
                              .bLimitBackwardEnable:=TIIB[EL7041-1000_M1L0_PitchCoarse]^STM Status^Status^Digital input 2;
                              .nRawEncoderULINT:=TIIB[EL5042_M1L0_PitchBender]^FB Inputs Channel 1^Position'}
    {attribute 'pytmc' := '
        pv: MR1L0:HOMS:MMS:PITCH
    '}
    M5 : ST_MotionStage := (fVelocity:=150.0,nEnableMode:=ENUM_StageEnableMode.ALWAYS, bPowerSelf:=TRUE, sName:='MR1L0_PITCH'); // M1L0 Pitch Stepper
    fbMotionStage_m5 : FB_MotionStage;

    {attribute 'TcLinkTo' := '.bLimitForwardEnable:=TIIB[EL7041-1000_M1L0_Bender]^STM Status^Status^Digital input 1;
                              .bLimitBackwardEnable:=TIIB[EL7041-1000_M1L0_Bender]^STM Status^Status^Digital input 2;
                              .nRawEncoderULINT:=TIIB[EL5042_M1L0_PitchBender]^FB Inputs Channel 2^Position'}
    {attribute 'pytmc' := '
        pv: MR1L0:HOMS:MMS:BENDER
    '}
    M6 : ST_MotionStage := (fVelocity:=150.0, nEnableMode:=ENUM_StageEnableMode.ALWAYS, bPowerSelf:=TRUE, sName:='MR1L0_BENDER'); // M1L0 Bender
    fbMotionStage_m6 : FB_MotionStage;

    {attribute 'TcLinkTo' := '.fbRunHOMS.bSTOEnable1:=TIIB[EL1004_M1L0_STO]^Channel 1^Input;
                              .fbRunHOMS.bSTOEnable2:=TIIB[EL1004_M1L0_STO]^Channel 2^Input;
                              .fbRunHOMS.stYupEnc.Count:=TIIB[EL5042_M1L0_Yupdwn]^FB Inputs Channel 1^Position;
                              .fbRunHOMS.stYdwnEnc.Count:=TIIB[EL5042_M1L0_Yupdwn]^FB Inputs Channel 2^Position;
                              .fbRunHOMS.stXupEnc.Count:=TIIB[EL5042_M1L0_Xupdwn]^FB Inputs Channel 1^Position;
                              .fbRunHOMS.stXdwnEnc.Count:=TIIB[EL5042_M1L0_Xupdwn]^FB Inputs Channel 2^Position'}
    {attribute 'pytmc' := '
        pv: MR1L0:HOMS
    '}
    M1L0 : DUT_HOMS;
    {attribute 'pytmc' := '
        pv: MR1L0:HOMS:STATS
    '}
    fbMR1L0GantryStats : FB_HomsStats;

    // Encoder Arrays/RMS Watch:
    {attribute 'pytmc' := '
        pv: MR1L0:HOMS:ENC:Y
    '}
    fbYRMSErrorM1L0 : FB_RMSWatch;
    fMaxYRMSErrorM1L0 : LREAL;
    fMinYRMSErrorM1L0 : LREAL;

    {attribute 'pytmc' := '
        pv: MR1L0:HOMS:ENC:X
    '}
    fbXRMSErrorM1L0 : FB_RMSWatch;
    fMaxXRMSErrorM1L0 : LREAL;
    fMinXRMSErrorM1L0 : LREAL;

    {attribute 'pytmc' := '
        pv: MR1L0:HOMS:ENC:PITCH
    '}
    fbPitchRMSErrorM1L0 : FB_RMSWatch;
    fMaxPitchRMSErrorM1L0 : LREAL;
    fMinPitchRMSErrorM1L0 : LREAL;

    {attribute 'pytmc' := '
        pv: MR1L0:HOMS:ENC:BENDER
    '}
    fbBenderRMSErrorM1L0 : FB_RMSWatch;
    fMaxBenderRMSErrorM1L0 : LREAL;
    fMinBenderRMSErrorM1L0 : LREAL;

    // Pitch Control
    //fbM1L0PitchControl : FB_PitchControl;
    //bM1L0PitchDone : BOOL;
    //bM1L0PitchBusy : BOOL;

    // Bender Control
    fbBenderM1L0 : FB_Bender;

    // Raw Encoder Counts
    {attribute 'pytmc' := '
        pv: MR1L0:HOMS:ENC:YUP:CNT
        field: EGU cnt
        io: i
    '}
    nEncCntYupM1L0 : UDINT;
    {attribute 'pytmc' := '
        pv: MR1L0:HOMS:ENC:YDWN:CNT
        field: EGU cnt
        io: i
    '}
    nEncCntYdwnM1L0 : UDINT;
    {attribute 'pytmc' := '
        pv: MR1L0:HOMS:ENC:XUP:CNT
        field: EGU cnt
        io: i
    '}
    nEncCntXupM1L0 : UDINT;
    {attribute 'pytmc' := '
        pv: MR1L0:HOMS:ENC:XDWN:CNT
        field: EGU cnt
        io: i
    '}
    nEncCntXdwnM1L0 : UDINT;
    {attribute 'pytmc' := '
        pv: MR1L0:HOMS:ENC:PITCH:CNT
        field: EGU cnt
        io: i
    '}
    nEncCntPitchM1L0 : UDINT;

    // Encoder Reference Values
    {attribute 'pytmc' := '
        pv: MR1L0:HOMS:ENC:YUP:REF
        field: EGU cnt
        io: i
    '}
    nEncRefYupM1L0 : UDINT;
    {attribute 'pytmc' := '
        pv: MR1L0:HOMS:ENC:YDWN:REF
        field: EGU cnt
        io: i
    '}
    nEncRefYdwnM1L0 : UDINT;
    {attribute 'pytmc' := '
        pv: MR1L0:HOMS:ENC:XUP:REF
        field: EGU cnt
        io: i
    '}
    nEncRefXupM1L0 : UDINT;
    {attribute 'pytmc' := '
        pv: MR1L0:HOMS:ENC:XDWN:REF
        field: EGU cnt
        io: i
    '}
    nEncRefXdwnM1L0 : UDINT;
    {attribute 'pytmc' := '
        pv: MR1L0:HOMS:ENC:PITCH:REF
        field: EGU cnt
        io: i
    '}
    nEncRefPitchM1L0 : UDINT;
    mcReadParameterPitchM1L0 : MC_ReadParameter;
    fEncRefPitchM1L0_urad : LREAL; // Current Pitch encoder offset in urad


    // M2L0
    // Motors
    {attribute 'TcLinkTo' := '.bLimitForwardEnable:=TIIB[EL7041-1000_M2L0_Yup]^STM Status^Status^Digital input 1;
                              .bLimitBackwardEnable:=TIIB[EL7041-1000_M2L0_Yup]^STM Status^Status^Digital input 2;
                              .nRawEncoderULINT:=TIIB[EL5042_M2L0_Yupdwn]^FB Inputs Channel 1^Position'}
    {attribute 'pytmc' := '
        pv: MR2L0:HOMS:MMS:YUP
    '}
    M7 : ST_MotionStage := (fVelocity:=200.0, nEnableMode:=ENUM_StageEnableMode.ALWAYS, bPowerSelf:=TRUE, sName:='MR2L0_YUP'); // M2L0 Yup
    fbMotionStage_m7 : FB_MotionStage;

    {attribute 'TcLinkTo' := '.bLimitForwardEnable:=TIIB[EL7041-1000_M2L0_Ydwn]^STM Status^Status^Digital input 1;
                              .bLimitBackwardEnable:=TIIB[EL7041-1000_M2L0_Ydwn]^STM Status^Status^Digital input 2'}
    {attribute 'pytmc' := '
        pv: MR2L0:HOMS:MMS:YDWN
    '}
    M8 : ST_MotionStage := (fVelocity:=200.0, nEnableMode:=ENUM_StageEnableMode.ALWAYS, bPowerSelf:=TRUE, sName:='MR2L0_YDWN'); // M2L0 Ydwn
    fbMotionStage_m8 : FB_MotionStage;

    {attribute 'TcLinkTo' := '.bLimitForwardEnable:=TIIB[EL7041-1000_M2L0_Xup]^STM Status^Status^Digital input 1;
                              .bLimitBackwardEnable:=TIIB[EL7041-1000_M2L0_Xup]^STM Status^Status^Digital input 2;
                              .nRawEncoderULINT:=TIIB[EL5042_M1L0_Xupdwn]^FB Inputs Channel 1^Position'}
    {attribute 'pytmc' := '
        pv: MR2L0:HOMS:MMS:XUP
    '}
    M9 : ST_MotionStage := (fVelocity:=1000.0, nEnableMode:=ENUM_StageEnableMode.ALWAYS, bPowerSelf:=TRUE, sName:='MR2L0_XUP'); // M2L0 Xup
    fbMotionStage_m9 : FB_MotionStage;

    {attribute 'TcLinkTo' := '.bLimitForwardEnable:=TIIB[EL7041-1000_M2L0_Xdwn]^STM Status^Status^Digital input 1;
                              .bLimitBackwardEnable:=TIIB[EL7041-1000_M2L0_Xdwn]^STM Status^Status^Digital input 2'}
    {attribute 'pytmc' := '
        pv: MR2L0:HOMS:MMS:XDWN
    '}
    M10 : ST_MotionStage := (fVelocity:=1000.0, nEnableMode:=ENUM_StageEnableMode.ALWAYS, bPowerSelf:=TRUE, sName:='MR2L0_XDWN'); // M2L0 Xdwn
    fbMotionStage_m10 : FB_MotionStage;

    {attribute 'TcLinkTo' := '.bLimitForwardEnable:=TIIB[EL7041-1000_M2L0_PitchCoarse]^STM Status^Status^Digital input 1;
                              .bLimitBackwardEnable:=TIIB[EL7041-1000_M2L0_PitchCoarse]^STM Status^Status^Digital input 2;
                              .nRawEncoderULINT:=TIIB[EL5042_M2L0_PitchBender]^FB Inputs Channel 1^Position'}
    {attribute 'pytmc' := '
        pv: MR2L0:HOMS:MMS:PITCH
    '}
    M11 : ST_MotionStage := (fVelocity:=150.0, nEnableMode:=ENUM_StageEnableMode.ALWAYS, bPowerSelf:=TRUE, sName:='MR2L0_PITCH'); // M2L0 Pitch Stepper
    fbMotionStage_m11 : FB_MotionStage;
    {attribute 'TcLinkTo' := '.bLimitForwardEnable:=TIIB[EL7041-1000_M2L0_Bender]^STM Status^Status^Digital input 1;
                              .bLimitBackwardEnable:=TIIB[EL7041-1000_M2L0_Bender]^STM Status^Status^Digital input 2;
                              .nRawEncoderULINT:=TIIB[EL5042_M2L0_PitchBender]^FB Inputs Channel 2^Position'}
    {attribute 'pytmc' := '
        pv: MR2L0:HOMS:MMS:BENDER
    '}
    M12 : ST_MotionStage := (fVelocity:=150.0, nEnableMode:=ENUM_StageEnableMode.ALWAYS, bPowerSelf:=TRUE, sName:='MR2L0_BENDER'); // M2L0 Bender
    fbMotionStage_m12 : FB_MotionStage;

    {attribute 'TcLinkTo' := '.fbRunHOMS.bSTOEnable1:=TIIB[EL1004_M2L0_STO]^Channel 1^Input;
                              .fbRunHOMS.bSTOEnable2:=TIIB[EL1004_M2L0_STO]^Channel 2^Input;
                              .fbRunHOMS.stYupEnc.Count:=TIIB[EL5042_M2L0_Yupdwn]^FB Inputs Channel 1^Position;
                              .fbRunHOMS.stYdwnEnc.Count:=TIIB[EL5042_M2L0_Yupdwn]^FB Inputs Channel 2^Position;
                              .fbRunHOMS.stXupEnc.Count:=TIIB[EL5042_M2L0_Xupdwn]^FB Inputs Channel 1^Position;
                              .fbRunHOMS.stXdwnEnc.Count:=TIIB[EL5042_M2L0_Xupdwn]^FB Inputs Channel 2^Position'}
    {attribute 'pytmc' := '
        pv: MR2L0:HOMS
    '}
    M2L0 : DUT_HOMS;
    {attribute 'pytmc' := '
        pv: MR2L0:HOMS:STATS
    '}
    fbMR2L0GantryStats : FB_HomsStats;

    // Encoder Arrays/RMS Watch:
    {attribute 'pytmc' := '
        pv: MR2L0:HOMS:ENC:Y
    '}
    fbYRMSErrorM2L0 : FB_RMSWatch;
    fMaxYRMSErrorM2L0 : LREAL;
    fMinYRMSErrorM2L0 : LREAL;

    {attribute 'pytmc' := '
        pv: MR2L0:HOMS:ENC:X
    '}
    fbXRMSErrorM2L0 : FB_RMSWatch;
    fMaxXRMSErrorM2L0 : LREAL;
    fMinXRMSErrorM2L0 : LREAL;

    {attribute 'pytmc' := '
        pv: MR2L0:HOMS:ENC:PITCH
    '}
    fbPitchRMSErrorM2L0 : FB_RMSWatch;
    fMaxPitchRMSErrorM2L0 : LREAL;
    fMinPitchRMSErrorM2L0 : LREAL;

    {attribute 'pytmc' := '
        pv: MR2L0:HOMS:ENC:BENDER
    '}
    fbBenderRMSErrorM2L0 : FB_RMSWatch;
    fMaxBenderRMSErrorM2L0 : LREAL;
    fMinBenderRMSErrorM2L0 : LREAL;

    // Pitch Control
    //fbM2L0PitchControl : FB_PitchControl;
    //bM2L0PitchDone : BOOL;
    //bM2L0PitchBusy : BOOL;

    // Bender Control
    fbBenderM2L0 : FB_Bender;

    // Raw Encoder Counts
    {attribute 'pytmc' := '
        pv: MR2L0:HOMS:ENC:YUP:CNT
        field: EGU cnt
        io: i
    '}
    nEncCntYupM2L0 : UDINT;
    {attribute 'pytmc' := '
        pv: MR2L0:HOMS:ENC:YDWN:CNT
        field: EGU cnt
        io: i
    '}
    nEncCntYdwnM2L0 : UDINT;
    {attribute 'pytmc' := '
        pv: MR2L0:HOMS:ENC:XUP:CNT
        field: EGU cnt
        io: i
    '}
    nEncCntXupM2L0 : UDINT;
    {attribute 'pytmc' := '
        pv: MR2L0:HOMS:ENC:XDWN:CNT
        field: EGU cnt
        io: i
    '}
    nEncCntXdwnM2L0 : UDINT;
    {attribute 'pytmc' := '
        pv: MR2L0:HOMS:ENC:PITCH:CNT
        field: EGU cnt
        io: i
    '}
    nEncCntPitchM2L0 : UDINT;

    // Encoder Reference Values
    {attribute 'pytmc' := '
        pv: MR2L0:HOMS:ENC:YUP:REF
        field: EGU cnt
        io: i
    '}
    nEncRefYupM2L0 : UDINT;
    {attribute 'pytmc' := '
        pv: MR2L0:HOMS:ENC:YDWN:REF
        field: EGU cnt
        io: i
    '}
    nEncRefYdwnM2L0 : UDINT;
    {attribute 'pytmc' := '
        pv: MR2L0:HOMS:ENC:XUP:REF
        field: EGU cnt
        io: i
    '}
    nEncRefXupM2L0 : UDINT;
    {attribute 'pytmc' := '
        pv: MR2L0:HOMS:ENC:XDWN:REF
        field: EGU cnt
        io: i
    '}
    nEncRefXdwnM2L0 : UDINT;
    {attribute 'pytmc' := '
        pv: MR2L0:HOMS:ENC:PITCH:REF
        field: EGU cnt
        io: i
    '}
    nEncRefPitchM2L0 : UDINT;
    mcReadParameterPitchM2L0 : MC_ReadParameter;
    fEncRefPitchM2L0_urad : LREAL; // Current Pitch encoder offset in urad

    //SP1L0:DCCM
    // Motors

    {attribute 'TcLinkTo' := '.bLimitForwardEnable:= TIIB[EL7047_SP1L0_th1]^STM Status^Status^Digital input 1;
                              .bLimitBackwardEnable:= TIIB[EL7047_SP1L0_th1]^STM Status^Status^Digital input 2;
                              .nRawEncoderULINT := TIIB[EL5042_SP1L0_th1_th2]^FB Inputs Channel 1^Position;'}
    {attribute 'pytmc' := '
        pv: SP1L0:DCCM:MMS:TH1
    '}
    M13 : ST_MotionStage := (nEnableMode:=ENUM_StageEnableMode.ALWAYS, bPowerSelf:=TRUE); // DCCM th1
    fbMotionStage_m13 : FB_MotionStage;

    {attribute 'TcLinkTo' := '.bLimitForwardEnable:= TIIB[EL7047_SP1L0_th2]^STM Status^Status^Digital input 1;
                              .bLimitBackwardEnable:= TIIB[EL7047_SP1L0_th2]^STM Status^Status^Digital input 2;
                              .nRawEncoderULINT := TIIB[EL5042_SP1L0_th1_th2]^FB Inputs Channel 2^Position;'}
    {attribute 'pytmc' := '
        pv: SP1L0:DCCM:MMS:TH2
    '}
    M14 : ST_MotionStage := (nEnableMode:=ENUM_StageEnableMode.ALWAYS, bPowerSelf:=TRUE); // DCCM th2
    fbMotionStage_m14 : FB_MotionStage;

    {attribute 'TcLinkTo' := '.bLimitForwardEnable:= TIIB[EL7047_SP1L0_tx]^STM Status^Status^Digital input 1;
                              .bLimitBackwardEnable:= TIIB[EL7047_SP1L0_tx]^STM Status^Status^Digital input 2;
                              .nRawEncoderULINT := TIIB[EL5042_SP1L0_tx_txd]^FB Inputs Channel 1^Position;'}
    {attribute 'pytmc' := '
        pv: SP1L0:DCCM:MMS:TX
    '}
    M15 : ST_MotionStage := (nEnableMode:=ENUM_StageEnableMode.ALWAYS, bPowerSelf:=TRUE); // DCCM tx
    fbMotionStage_m15 : FB_MotionStage;

    {attribute 'TcLinkTo' := '.bLimitForwardEnable:= TIIB[EL7047_SP1L0_txd]^STM Status^Status^Digital input 1;
                              .bLimitBackwardEnable:= TIIB[EL7047_SP1L0_txd]^STM Status^Status^Digital input 2;
                              .nRawEncoderULINT := TIIB[EL5042_SP1L0_tx_txd]^FB Inputs Channel 2^Position;'}
    {attribute 'pytmc' := '
        pv: SP1L0:DCCM:MMS:TXD
    '}
    M16 : ST_MotionStage := (nEnableMode:=ENUM_StageEnableMode.ALWAYS, bPowerSelf:=TRUE); // DCCM txd
    fbMotionStage_m16 : FB_MotionStage;

    {attribute 'TcLinkTo' := '.bLimitForwardEnable:= TIIB[EL7047_SP1L0_tyd]^STM Status^Status^Digital input 1;
                              .bLimitBackwardEnable:= TIIB[EL7047_SP1L0_tyd]^STM Status^Status^Digital input 2;
                              .nRawEncoderULINT := TIIB[EL5042_SP1L0_tyd]^FB Inputs Channel 1^Position;'}
    {attribute 'pytmc' := '
        pv: SP1L0:DCCM:MMS:TYD
    '}
    M17 : ST_MotionStage := (nEnableMode:=ENUM_StageEnableMode.ALWAYS, bPowerSelf:=TRUE); // DCCM tyd
    fbMotionStage_m17 : FB_MotionStage;

 //Analog input for Tx Brake Pressure Sensor. Sensor to monitor pressure to verify brakes are released. 90PSI to release brakes.

    {attribute 'pytmc' := '
        pv: DCCM:MONO:SOL
    '}
    {attribute 'TcLinkTo' :='TIIB[EL3054_SP1L0_AI]^AI Standard Channel 1^Value'}
    nAI AT %I*:UINT;

//digital outputs
//DO for Compressed Air Solenoid Actuation on Tx to release brake. Brakes released when pressure is applied.
      {attribute 'pytmc' := '
        pv: SP1L0:DCCM:TX:BRAKE
        field: ZNAM OFF ;
        field: ONAM ON ;
    '}
     {attribute 'TcLinkTo' := 'TIIB[EL2008_SP1L0_DO]^Channel 1^Output'}
    bTx_Brake_Solenoid AT %Q*:BOOL;

       {attribute 'pytmc' := '
        pv: SP1L0:DCCM:DO1
        field: ZNAM OFF ;
        field: ONAM ON ;
    '}
     {attribute 'TcLinkTo' := 'TIIB[EL2008_SP1L0_DO]^Channel 2^Output'}
    bDO1 AT %Q*:BOOL;

       {attribute 'pytmc' := '
        pv: SP1L0:DCCM:DO2
        field: ZNAM OFF ;
        field: ONAM ON ;
    '}
     {attribute 'TcLinkTo' := 'TIIB[EL2008_SP1L0_DO]^Channel 3^Output'}
    bDO2 AT %Q*:BOOL;

         {attribute 'pytmc' := '
        pv: SP1L0:DCCM:DO3
        field: ZNAM OFF ;
        field: ONAM ON ;
    '}
     {attribute 'TcLinkTo' := 'TIIB[EL2008_SP1L0_DO]^Channel 4^Output'}
    bDO3 AT %Q*:BOOL;

         {attribute 'pytmc' := '
        pv: SP1L0:DCCM:DO4
        field: ZNAM OFF ;
        field: ONAM ON ;
    '}
     {attribute 'TcLinkTo' := 'TIIB[EL2008_SP1L0_DO]^Channel 5^Output'}
    bDO4 AT %Q*:BOOL;

         {attribute 'pytmc' := '
        pv: SP1L0:DCCM:DO5
        field: ZNAM OFF ;
        field: ONAM ON ;
    '}
     {attribute 'TcLinkTo' := 'TIIB[EL2008_SP1L0_DO]^Channel 6^Output'}
    bDO5 AT %Q*:BOOL;

         {attribute 'pytmc' := '
        pv: SP1L0:DCCM:DO6
        field: ZNAM OFF ;
        field: ONAM ON ;
    '}
     {attribute 'TcLinkTo' := 'TIIB[EL2008_SP1L0_DO]^Channel 7^Output'}
    bDO6 AT %Q*:BOOL;

        {attribute 'pytmc' := '
        pv: SP1L0:DCCM:FAN:PWR
        field: ZNAM OFF ;
        field: ONAM ON ;
    '}
     {attribute 'TcLinkTo' := 'TIIB[EL2008_SP1L0_DO]^Channel 8^Output'}
    bFanOn AT %Q*:BOOL;

(* digital inputs, 6x overtravel limits, 1x STO, 1x spare *)

    {attribute 'pytmc' := '
        pv: SP1L0:DCCM:TH1:POTL
        field: ZNAM OFF ;
        field: ONAM ON ;
    '}
    {attribute 'TcLinkTo' := 'TIIB[EL1008_SP1L0_STO_DI]^Channel 1^Input'}
    bTH1_POTL AT %I*:BOOL;

        {attribute 'pytmc' := '
        pv: SP1L0:DCCM:TH1:NOTL
        field: ZNAM OFF ;
        field: ONAM ON ;
    '}
    {attribute 'TcLinkTo' := 'TIIB[EL1008_SP1L0_STO_DI]^Channel 2^Input'}
    bTH1_NOTL AT %I*:BOOL;

    {attribute 'pytmc' := '
        pv: SP1L0:DCCM:TH2:POTL
        field: ZNAM OFF ;
        field: ONAM ON ;
    '}
    {attribute 'TcLinkTo' := 'TIIB[EL1008_SP1L0_STO_DI]^Channel 3^Input'}
    bTH2_POTL AT %I*:BOOL;

        {attribute 'pytmc' := '
        pv: SP1L0:DCCM:TH2:NOTL
        field: ZNAM OFF ;
        field: ONAM ON ;
    '}
    {attribute 'TcLinkTo' := 'TIIB[EL1008_SP1L0_STO_DI]^Channel 4^Input'}
    bTH2_NOTL AT %I*:BOOL;

        {attribute 'pytmc' := '
        pv: SP1L0:DCCM:TX:POTL
        field: ZNAM OFF ;
        field: ONAM ON ;
    '}
    {attribute 'TcLinkTo' := 'TIIB[EL1008_SP1L0_STO_DI]^Channel 5^Input'}
    bTX_POTL AT %I*:BOOL;

        {attribute 'pytmc' := '
        pv: SP1L0:DCCM:TX:NOTL
        field: ZNAM OFF ;
        field: ONAM ON ;
    '}
    {attribute 'TcLinkTo' := 'TIIB[EL1008_SP1L0_STO_DI]^Channel 6^Input'}
    bTX_NOTL AT %I*:BOOL;


    {attribute 'pytmc' := '
        pv: SP1L0:DCCM:STO
        field: ZNAM OFF ;
        field: ONAM ON ;
    '}
    {attribute 'TcLinkTo' := 'TIIB[EL1008_SP1L0_STO_DI]^Channel 7^Input'}
    bSTO AT %I*:BOOL;

    {attribute 'pytmc' := '
        pv: SP1L0:DCCM:DI7
        field: ZNAM OFF ;
        field: ONAM ON ;
    '}
    {attribute 'TcLinkTo' := 'TIIB[EL1008_SP1L0_STO_DI]^Channel 8^Input'}
    bDI7 AT %I*:BOOL;

    // Common
    fEncLeverArm_mm : LREAL := 513.0;
    // Logging
    fbLogHandler : FB_LogHandler;

END_VAR

// M1L0
M1L0.fbRunHOMS(stYup:=M1,
               stYdwn:=M2,
               stXup:=M3,
               stXdwn:=M4,
               stPitch:=M5,
               nYupEncRef:=GVL_M1L0_Constants.nYUP_ENC_REF,
               nYdwnEncRef:=GVL_M1L0_Constants.nYDWN_ENC_REF,
               nXupEncRef:=GVL_M1L0_Constants.nXUP_ENC_REF,
               nXdwnEncRef:=GVL_M1L0_Constants.nXDWN_ENC_REF,
               bExecuteCoupleY:=M1L0.bExecuteCoupleY,
               bExecuteCoupleX:=M1L0.bExecuteCoupleX,
               bExecuteDecoupleY:=M1L0.bExecuteDecoupleY,
               bExecuteDecoupleX:=M1L0.bExecuteDecoupleX,
               bGantryAlreadyCoupledY=>M1L0.bGantryAlreadyCoupledY,
               bGantryAlreadyCoupledX=>M1L0.bGantryAlreadyCoupledX,
               nCurrGantryY=>M1L0.nCurrGantryY,
               nCurrGantryX=>M1L0.nCurrGantryX);
fbBenderM1L0(stBender:=M6,
             bSTOEnable1:=M1L0.fbRunHOMS.bSTOEnable1,
             bSTOEnable2:=M1L0.fbRunHOMS.bSTOEnable2);
// No slave motion through Epics
M2.bExecute := FALSE; // M1L0-Ydwn
M4.bExecute := FALSE; // M1L0-Xdwn

// Convert nCurrGantry to um (smaller number) to read out in epics
M1L0.fCurrGantryY_um := LINT_TO_REAL(M1L0.nCurrGantryY) / 1000.0;
M1L0.fCurrGantryX_um := LINT_TO_REAL(M1L0.nCurrGantryX) / 1000.0;

// FB_MotionStage's for non-piezo axes
fbMotionStage_m1(stMotionStage:=M1);
fbMotionStage_m2(stMotionStage:=M2);
fbMotionStage_m3(stMotionStage:=M3);
fbMotionStage_m4(stMotionStage:=M4);
fbMotionStage_m5(stMotionStage:=M5);
fbMotionStage_m6(stMotionStage:=M6);

// Calulate Gantry Stats:
fbMR1L0GantryStats(homs:=M1L0, fbUpStreamY:=M1, fbUpStreamX:=M3);
fbMR2L0GantryStats(homs:=M2L0, fbUpStreamY:=M7, fbUpStreamX:=M9);


// Calculate Pitch RMS Error:
fbYRMSErrorM1L0(stMotionStage:=M1,
                fMaxRMSError=>fMaxYRMSErrorM1L0,
                fMinRMSError=>fMinYRMSErrorM1L0);

fbXRMSErrorM1L0(stMotionStage:=M3,
                fMaxRMSError=>fMaxXRMSErrorM1L0,
                fMinRMSError=>fMinXRMSErrorM1L0);

fbPitchRMSErrorM1L0(stMotionStage:=M5,
                    fMaxRMSError=>fMaxPitchRMSErrorM1L0,
                    fMinRMSError=>fMinPitchRMSErrorM1L0);

fbBenderRMSErrorM1L0(stMotionStage:=M6,
                     fMaxRMSError=>fMaxBenderRMSErrorM1L0,
                     fMinRMSError=>fMinBenderRMSErrorM1L0);
// Pitch Control
//fbM1L0PitchControl(Pitch:=GVL_M1L0.M1L0_Pitch,
                   //Stepper:=M5,
                   //lrCurrentSetpoint:=M5.fPosition,
                   //q_bDone=>bM1L0PitchDone,
                   //q_bBusy=>bM1L0PitchBusy);
// When STO hit, need to reset SP
//IF NOT M5.bHardwareEnable THEN
    //M5.fPosition := M5.stAxisStatus.fActPosition;
//END_IF

// Raw Encoder Counts For Epics
nEncCntYupM1L0 := ULINT_TO_UDINT(M1L0.fbRunHOMS.stYupEnc.Count);
nEncCntYdwnM1L0 := ULINT_TO_UDINT(M1L0.fbRunHOMS.stYdwnEnc.Count);
nEncCntXupM1L0 := ULINT_TO_UDINT(M1L0.fbRunHOMS.stXupEnc.Count);
nEncCntXdwnM1L0 := ULINT_TO_UDINT(M1L0.fbRunHOMS.stXdwnEnc.Count);
nEncCntPitchM1L0 := LINT_TO_UDINT(GVL_M1L0.M1L0_Pitch.diEncCnt);

// Encoder Reference Values For Epics
nEncRefYupM1L0 := ULINT_TO_UDINT(GVL_M1L0_Constants.nYUP_ENC_REF);
nEncRefYdwnM1L0 := ULINT_TO_UDINT(GVL_M1L0_Constants.nYDWN_ENC_REF);
nEncRefXupM1L0 := ULINT_TO_UDINT(GVL_M1L0_Constants.nXUP_ENC_REF);
nEncRefXdwnM1L0 := ULINT_TO_UDINT(GVL_M1L0_Constants.nXDWN_ENC_REF);
mcReadParameterPitchM1L0(Axis:=M5.Axis,
                         Enable:=TRUE,
                         ParameterNumber:=MC_AxisParameter.AxisEncoderOffset,
                         ReadMode:=READMODE_CYCLIC,
                         Value=>fEncRefPitchM1L0_urad);

nEncRefPitchM1L0 := LREAL_TO_UDINT(ABS(fEncRefPitchM1L0_urad) * fEncLeverArm_mm);

//Coatings States With PMPS
M1.bPowerSelf :=FALSE;
M5.bPowerSelf := FALSE;




// M2L0
M2L0.fbRunHOMS(stYup:=M7,
               stYdwn:=M8,
               stXup:=M9,
               stXdwn:=M10,
               stPitch:=M11,
               nYupEncRef:=GVL_M2L0_Constants.nYUP_ENC_REF,
               nYdwnEncRef:=GVL_M2L0_Constants.nYDWN_ENC_REF,
               nXupEncRef:=GVL_M2L0_Constants.nXUP_ENC_REF,
               nXdwnEncRef:=GVL_M2L0_Constants.nXDWN_ENC_REF,
               bExecuteCoupleY:=M2L0.bExecuteCoupleY,
               bExecuteCoupleX:=M2L0.bExecuteCoupleX,
               bExecuteDecoupleY:=M2L0.bExecuteDecoupleY,
               bExecuteDecoupleX:=M2L0.bExecuteDecoupleX,
               bGantryAlreadyCoupledY=>M2L0.bGantryAlreadyCoupledY,
               bGantryAlreadyCoupledX=>M2L0.bGantryAlreadyCoupledX,
               nCurrGantryY=>M2L0.nCurrGantryY,
               nCurrGantryX=>M2L0.nCurrGantryX);
fbBenderM2L0(stBender:=M12,
             bSTOEnable1:=M2L0.fbRunHOMS.bSTOEnable1,
             bSTOEnable2:=M2L0.fbRunHOMS.bSTOEnable2);
// No slave motion through Epics
M8.bExecute := FALSE; // M2L0-Ydwn
M10.bExecute := FALSE; // M2L0-Xdwn

